LIN {X 0,Y 474.601,Z 136.99,A -85,B 0,C 180,E1 -7407.326,E2 -7407.326} C_VEL
LIN {X 0,Y 474.598,Z 136.978,A -85,B 0,C 180,E1 -7410.231,E2 -7410.231} C_VEL
LIN {X 0,Y 474.615,Z 136.966,A -85,B 0,C 180,E1 -7413.222,E2 -7413.222} C_VEL
LIN {X 0,Y 474.584,Z 136.991,A -85,B 0,C 180,E1 -7416.324,E2 -7416.324} C_VEL
LIN {X 0,Y 474.622,Z 136.969,A -85,B 0,C 180,E1 -7419.548,E2 -7419.548} C_VEL
LIN {X 0,Y 474.577,Z 136.989,A -85,B 0,C 180,E1 -7422.23,E2 -7422.23} C_VEL
LIN {X 0,Y 474.616,Z 136.982,A -85,B 0,C 180,E1 -7425.298,E2 -7425.298} C_VEL
LIN {X 0,Y 474.592,Z 136.991,A -85,B 0,C 180,E1 -7428.211,E2 -7428.211} C_VEL
LIN {X 0,Y 474.608,Z 136.991,A -85,B 0,C 180,E1 -7431.542,E2 -7431.542} C_VEL
LIN {X 0,Y 474.617,Z 136.989,A -85,B 0,C 180,E1 -7434.725,E2 -7434.725} C_VEL
LIN {X 0,Y 474.629,Z 136.988,A -85,B 0,C 180,E1 -7437.787,E2 -7437.787} C_VEL
LIN {X 0,Y 474.575,Z 136.983,A -85,B 0,C 180,E1 -7440.896,E2 -7440.896} C_VEL
LIN {X 0,Y 474.643,Z 137.123,A -85,B 0,C 180,E1 -7442.017,E2 -7442.017} C_VEL
LIN {X 0,Y 477.053,Z 147.679,A -85,B 0,C 180,E1 -7443.983,E2 -7443.983} C_VEL
LIN {X 0,Y 478.463,Z 154.908,A -85,B 0,C 180,E1 -7445.252,E2 -7445.252} C_VEL
LIN {X 0,Y 478.125,Z 161.386,A -85,B 0,C 180,E1 -7446.26,E2 -7446.26} C_VEL
LIN {X 0,Y 479.797,Z 169.232,A -85,B 0,C 180,E1 -7446.509,E2 -7446.509} C_VEL
LIN {X 0,Y 482.553,Z 182.514,A -85,B 0,C 180,E1 -7446.862,E2 -7446.862} C_VEL
LIN {X 0,Y 482.481,Z 187.574,A -85,B 0,C 180,E1 -7446.939,E2 -7446.939} C_VEL
LIN {X 0,Y 481.775,Z 193.424,A -85,B 0,C 180,E1 -7446.996,E2 -7446.996} C_VEL
LIN {X 0,Y 476.297,Z 212.491,A -85,B 0,C 180,E1 -7447.021,E2 -7447.021} C_VEL
LIN {X 0,Y 475.613,Z 218.341,A -85,B 0,C 180,E1 -7447.08,E2 -7447.08} C_VEL
LIN {X 0,Y 474.357,Z 326.967,A -85,B 0,C 180,E1 -7448.779,E2 -7448.779} C_VEL
LIN {X 0,Y 473.824,Z 342.596,A -85,B 0,C 180,E1 -7449.193,E2 -7449.193} C_VEL
LIN {X 0,Y 473.371,Z 356.882,A -85,B 0,C 180,E1 -7449.749,E2 -7449.749} C_VEL
LIN {X 0,Y 472.578,Z 370.807,A -85,B 0,C 180,E1 -7450.451,E2 -7450.451} C_VEL
LIN {X 0,Y 471.793,Z 384.429,A -85,B 0,C 180,E1 -7451.321,E2 -7451.321} C_VEL
LIN {X 0,Y 470.896,Z 396.958,A -85,B 0,C 180,E1 -7452.296,E2 -7452.296} C_VEL
LIN {X 0,Y 470.076,Z 409.646,A -85,B 0,C 180,E1 -7453.497,E2 -7453.497} C_VEL
LIN {X 0,Y 469.269,Z 421.151,A -85,B 0,C 180,E1 -7454.806,E2 -7454.806} C_VEL
LIN {X 0,Y 468.595,Z 430.834,A -85,B 0,C 180,E1 -7456.115,E2 -7456.115} C_VEL
LIN {X 0,Y 467.975,Z 440.24,A -85,B 0,C 180,E1 -7457.627,E2 -7457.627} C_VEL
LIN {X 0,Y 467.546,Z 448.231,A -85,B 0,C 180,E1 -7459.17,E2 -7459.17} C_VEL
LIN {X 0,Y 467.105,Z 455.613,A -85,B 0,C 180,E1 -7460.91,E2 -7460.91} C_VEL
LIN {X 0,Y 466.844,Z 461.472,A -85,B 0,C 180,E1 -7462.648,E2 -7462.648} C_VEL
LIN {X 0,Y 466.79,Z 464.941,A -85,B 0,C 180,E1 -7463.95,E2 -7463.95} C_VEL
LIN {X 0,Y 466.625,Z 468.461,A -85,B 0,C 180,E1 -7465.681,E2 -7465.681} C_VEL
LIN {X 0,Y 466.657,Z 470.79,A -85,B 0,C 180,E1 -7467.41,E2 -7467.41} C_VEL
LIN {X 0,Y 466.587,Z 471.982,A -85,B 0,C 180,E1 -7469.137,E2 -7469.137} C_VEL
LIN {X 0,Y 466.587,Z 472,A -85,B 0,C 180,E1 -7470.863,E2 -7470.863} C_VEL
LIN {X 0,Y 466.658,Z 470.878,A -85,B 0,C 180,E1 -7472.59,E2 -7472.59} C_VEL
LIN {X 0,Y 466.624,Z 468.618,A -85,B 0,C 180,E1 -7474.319,E2 -7474.319} C_VEL
LIN {X 0,Y 466.763,Z 465.163,A -85,B 0,C 180,E1 -7476.05,E2 -7476.05} C_VEL
LIN {X 0,Y 466.909,Z 460.435,A -85,B 0,C 180,E1 -7477.786,E2 -7477.786} C_VEL
LIN {X 0,Y 467.191,Z 454.309,A -85,B 0,C 180,E1 -7479.525,E2 -7479.525} C_VEL
LIN {X 0,Y 467.659,Z 446.597,A -85,B 0,C 180,E1 -7481.266,E2 -7481.266} C_VEL
LIN {X 0,Y 468.093,Z 438.528,A -85,B 0,C 180,E1 -7482.768,E2 -7482.768} C_VEL
LIN {X 0,Y 468.775,Z 428.476,A -85,B 0,C 180,E1 -7484.322,E2 -7484.322} C_VEL
LIN {X 0,Y 469.43,Z 418.327,A -85,B 0,C 180,E1 -7485.634,E2 -7485.634} C_VEL
LIN {X 0,Y 470.225,Z 407.623,A -85,B 0,C 180,E1 -7486.801,E2 -7486.801} C_VEL
LIN {X 0,Y 471.044,Z 395.428,A -85,B 0,C 180,E1 -7487.922,E2 -7487.922} C_VEL
LIN {X 0,Y 471.888,Z 382.566,A -85,B 0,C 180,E1 -7488.901,E2 -7488.901} C_VEL
LIN {X 0,Y 472.684,Z 368.463,A -85,B 0,C 180,E1 -7489.771,E2 -7489.771} C_VEL
LIN {X 0,Y 473.487,Z 353.414,A -85,B 0,C 180,E1 -7490.489,E2 -7490.489} C_VEL
LIN {X 0,Y 473.958,Z 339.526,A -85,B 0,C 180,E1 -7490.99,E2 -7490.99} C_VEL
LIN {X 0,Y 474.358,Z 325.557,A -85,B 0,C 180,E1 -7491.341,E2 -7491.341} C_VEL
LIN {X 0,Y 476.011,Z 183.2,A -85,B 0,C 180,E1 -7493.558,E2 -7493.558} C_VEL
LIN {X 0,Y 471.382,Z 161.527,A -85,B 0,C 180,E1 -7494.186,E2 -7494.186} C_VEL
LIN {X 0,Y 471.552,Z 155.541,A -85,B 0,C 180,E1 -7495.136,E2 -7495.136} C_VEL
LIN {X 0,Y 468.023,Z 139.951,A -85,B 0,C 180,E1 -7497.986,E2 -7497.986} C_VEL
LIN {X 0,Y 467.569,Z 137.908,A -85,B 0,C 180,E1 -7498.444,E2 -7498.444} C_VEL
LIN {X 0,Y 467.546,Z 137.867,A -85,B 0,C 180,E1 -7501.743,E2 -7501.743} C_VEL
LIN {X 0,Y 467.551,Z 137.87,A -85,B 0,C 180,E1 -7504.834,E2 -7504.834} C_VEL
LIN {X 0,Y 467.541,Z 137.87,A -85,B 0,C 180,E1 -7508.047,E2 -7508.047} C_VEL
LIN {X 0,Y 467.561,Z 137.87,A -85,B 0,C 180,E1 -7511.274,E2 -7511.274} C_VEL
LIN {X 0,Y 467.566,Z 137.861,A -85,B 0,C 180,E1 -7514.948,E2 -7514.948} C_VEL
LIN {X 0,Y 467.559,Z 137.858,A -85,B 0,C 180,E1 -7518.595,E2 -7518.595} C_VEL
LIN {X 0,Y 467.552,Z 137.86,A -85,B 0,C 180,E1 -7521.411,E2 -7521.411} C_VEL
LIN {X 0,Y 467.558,Z 137.87,A -85,B 0,C 180,E1 -7524.262,E2 -7524.262} C_VEL
LIN {X 0,Y 467.575,Z 137.84,A -85,B 0,C 180,E1 -7527.323,E2 -7527.323} C_VEL
LIN {X 0,Y 467.552,Z 137.867,A -85,B 0,C 180,E1 -7530.672,E2 -7530.672} C_VEL
LIN {X 0,Y 467.536,Z 137.867,A -85,B 0,C 180,E1 -7533.195,E2 -7533.195} C_VEL
LIN {X 0,Y 467.557,Z 137.865,A -85,B 0,C 180,E1 -7536.056,E2 -7536.056} C_VEL
LIN {X 0,Y 467.621,Z 137.855,A -85,B 0,C 180,E1 -7539.777,E2 -7539.777} C_VEL
LIN {X 0,Y 467.57,Z 137.866,A -85,B 0,C 180,E1 -7542.505,E2 -7542.505} C_VEL
LIN {X 0,Y 467.596,Z 137.855,A -85,B 0,C 180,E1 -7545.196,E2 -7545.196} C_VEL
LIN {X 0,Y 467.659,Z 137.857,A -85,B 0,C 180,E1 -7547.855,E2 -7547.855} C_VEL
LIN {X 0,Y 467.669,Z 137.847,A -85,B 0,C 180,E1 -7551.357,E2 -7551.357} C_VEL
LIN {X 0,Y 467.723,Z 137.849,A -85,B 0,C 180,E1 -7553.962,E2 -7553.962} C_VEL
LIN {X 0,Y 467.824,Z 137.827,A -85,B 0,C 180,E1 -7557.417,E2 -7557.417} C_VEL
LIN {X 0,Y 467.881,Z 137.826,A -85,B 0,C 180,E1 -7560,E2 -7560} C_VEL
LIN {X 0,Y 467.852,Z 137.823,A -85,B 0,C 180,E1 -7562.583,E2 -7562.583} C_VEL
LIN {X 0,Y 467.725,Z 137.845,A -85,B 0,C 180,E1 -7566.038,E2 -7566.038} C_VEL
LIN {X 0,Y 467.671,Z 137.848,A -85,B 0,C 180,E1 -7568.643,E2 -7568.643} C_VEL
LIN {X 0,Y 467.658,Z 137.853,A -85,B 0,C 180,E1 -7572.145,E2 -7572.145} C_VEL
LIN {X 0,Y 467.64,Z 137.85,A -85,B 0,C 180,E1 -7575.695,E2 -7575.695} C_VEL
LIN {X 0,Y 467.623,Z 137.858,A -85,B 0,C 180,E1 -7579.308,E2 -7579.308} C_VEL
LIN {X 0,Y 467.536,Z 137.865,A -85,B 0,C 180,E1 -7582.074,E2 -7582.074} C_VEL
LIN {X 0,Y 467.58,Z 137.863,A -85,B 0,C 180,E1 -7584.889,E2 -7584.889} C_VEL
LIN {X 0,Y 467.618,Z 137.858,A -85,B 0,C 180,E1 -7587.769,E2 -7587.769} C_VEL
LIN {X 0,Y 467.568,Z 137.853,A -85,B 0,C 180,E1 -7591.044,E2 -7591.044} C_VEL
LIN {X 0,Y 467.577,Z 137.846,A -85,B 0,C 180,E1 -7594.24,E2 -7594.24} C_VEL
LIN {X 0,Y 467.549,Z 137.868,A -85,B 0,C 180,E1 -7597.186,E2 -7597.186} C_VEL
LIN {X 0,Y 467.578,Z 137.85,A -85,B 0,C 180,E1 -7600.264,E2 -7600.264} C_VEL
LIN {X 0,Y 467.587,Z 137.866,A -85,B 0,C 180,E1 -7602.567,E2 -7602.567} C_VEL
LIN {X 0,Y 467.567,Z 137.859,A -85,B 0,C 180,E1 -7605.052,E2 -7605.052} C_VEL
LIN {X 0,Y 467.59,Z 137.859,A -85,B 0,C 180,E1 -7607.44,E2 -7607.44} C_VEL
LIN {X 0,Y 467.561,Z 137.861,A -85,B 0,C 180,E1 -7610.853,E2 -7610.853} C_VEL
LIN {X 0,Y 467.56,Z 137.863,A -85,B 0,C 180,E1 -7614.261,E2 -7614.261} C_VEL
LIN {X 0,Y 467.582,Z 137.843,A -85,B 0,C 180,E1 -7617.321,E2 -7617.321} C_VEL
LIN {X 0,Y 467.593,Z 137.978,A -85,B 0,C 180,E1 -7620.582,E2 -7620.582} C_VEL
LIN {X 0,Y 470.698,Z 150.848,A -85,B 0,C 180,E1 -7622.909,E2 -7622.909} C_VEL
LIN {X 0,Y 471.908,Z 156.825,A -85,B 0,C 180,E1 -7623.938,E2 -7623.938} C_VEL
LIN {X 0,Y 471.272,Z 169.442,A -85,B 0,C 180,E1 -7625.859,E2 -7625.859} C_VEL
LIN {X 0,Y 475.948,Z 192.592,A -85,B 0,C 180,E1 -7626.504,E2 -7626.504} C_VEL
LIN {X 0,Y 474.317,Z 332.942,A -85,B 0,C 180,E1 -7628.686,E2 -7628.686} C_VEL
LIN {X 0,Y 473.837,Z 348.179,A -85,B 0,C 180,E1 -7629.062,E2 -7629.062} C_VEL
LIN {X 0,Y 473.282,Z 362.937,A -85,B 0,C 180,E1 -7629.601,E2 -7629.601} C_VEL
LIN {X 0,Y 472.605,Z 375.987,A -85,B 0,C 180,E1 -7630.226,E2 -7630.226} C_VEL
LIN {X 0,Y 471.76,Z 390.279,A -85,B 0,C 180,E1 -7631.094,E2 -7631.094} C_VEL
LIN {X 0,Y 470.911,Z 403.288,A -85,B 0,C 180,E1 -7632.072,E2 -7632.072} C_VEL
LIN {X 0,Y 470.149,Z 414.467,A -85,B 0,C 180,E1 -7633.078,E2 -7633.078} C_VEL
LIN {X 0,Y 469.274,Z 426.416,A -85,B 0,C 180,E1 -7634.361,E2 -7634.361} C_VEL
LIN {X 0,Y 468.65,Z 436.644,A -85,B 0,C 180,E1 -7635.674,E2 -7635.674} C_VEL
LIN {X 0,Y 467.949,Z 446.598,A -85,B 0,C 180,E1 -7637.194,E2 -7637.194} C_VEL
LIN {X 0,Y 467.589,Z 454.94,A -85,B 0,C 180,E1 -7638.732,E2 -7638.732} C_VEL
LIN {X 0,Y 467.104,Z 462.734,A -85,B 0,C 180,E1 -7640.473,E2 -7640.473} C_VEL
LIN {X 0,Y 466.86,Z 468.934,A -85,B 0,C 180,E1 -7642.213,E2 -7642.213} C_VEL
LIN {X 0,Y 466.726,Z 473.728,A -85,B 0,C 180,E1 -7643.949,E2 -7643.949} C_VEL
LIN {X 0,Y 466.601,Z 477.239,A -85,B 0,C 180,E1 -7645.681,E2 -7645.681} C_VEL
LIN {X 0,Y 466.637,Z 479.55,A -85,B 0,C 180,E1 -7647.41,E2 -7647.41} C_VEL
LIN {X 0,Y 466.586,Z 480.712,A -85,B 0,C 180,E1 -7649.137,E2 -7649.137} C_VEL
LIN {X 0,Y 466.586,Z 480.711,A -85,B 0,C 180,E1 -7650.863,E2 -7650.863} C_VEL
LIN {X 0,Y 466.637,Z 479.545,A -85,B 0,C 180,E1 -7652.59,E2 -7652.59} C_VEL
LIN {X 0,Y 466.602,Z 477.233,A -85,B 0,C 180,E1 -7654.319,E2 -7654.319} C_VEL
LIN {X 0,Y 466.751,Z 473.727,A -85,B 0,C 180,E1 -7656.05,E2 -7656.05} C_VEL
LIN {X 0,Y 466.86,Z 468.935,A -85,B 0,C 180,E1 -7657.787,E2 -7657.787} C_VEL
LIN {X 0,Y 467.104,Z 462.726,A -85,B 0,C 180,E1 -7659.527,E2 -7659.527} C_VEL
LIN {X 0,Y 467.588,Z 454.928,A -85,B 0,C 180,E1 -7661.268,E2 -7661.268} C_VEL
LIN {X 0,Y 467.975,Z 446.451,A -85,B 0,C 180,E1 -7662.827,E2 -7662.827} C_VEL
LIN {X 0,Y 468.651,Z 436.633,A -85,B 0,C 180,E1 -7664.326,E2 -7664.326} C_VEL
LIN {X 0,Y 469.301,Z 426.404,A -85,B 0,C 180,E1 -7665.638,E2 -7665.638} C_VEL
LIN {X 0,Y 470.134,Z 414.519,A -85,B 0,C 180,E1 -7666.916,E2 -7666.916} C_VEL
LIN {X 0,Y 470.986,Z 401.979,A -85,B 0,C 180,E1 -7668.037,E2 -7668.037} C_VEL
LIN {X 0,Y 471.834,Z 388.66,A -85,B 0,C 180,E1 -7669.016,E2 -7669.016} C_VEL
LIN {X 0,Y 472.627,Z 375.945,A -85,B 0,C 180,E1 -7669.773,E2 -7669.773} C_VEL
LIN {X 0,Y 473.254,Z 362.971,A -85,B 0,C 180,E1 -7670.397,E2 -7670.397} C_VEL
LIN {X 0,Y 473.858,Z 348.12,A -85,B 0,C 180,E1 -7670.937,E2 -7670.937} C_VEL
LIN {X 0,Y 474.293,Z 332.817,A -85,B 0,C 180,E1 -7671.315,E2 -7671.315} C_VEL
LIN {X 0,Y 475.947,Z 192.412,A -85,B 0,C 180,E1 -7673.496,E2 -7673.496} C_VEL
LIN {X 0,Y 471.259,Z 169.525,A -85,B 0,C 180,E1 -7674.133,E2 -7674.133} C_VEL
LIN {X 0,Y 471.878,Z 156.807,A -85,B 0,C 180,E1 -7676.063,E2 -7676.063} C_VEL
LIN {X 0,Y 469.216,Z 144.362,A -85,B 0,C 180,E1 -7678.23,E2 -7678.23} C_VEL
LIN {X 0,Y 467.581,Z 137.946,A -85,B 0,C 180,E1 -7679.434,E2 -7679.434} C_VEL
LIN {X 0,Y 467.584,Z 137.845,A -85,B 0,C 180,E1 -7682.758,E2 -7682.758} C_VEL
LIN {X 0,Y 467.554,Z 137.864,A -85,B 0,C 180,E1 -7685.89,E2 -7685.89} C_VEL
LIN {X 0,Y 467.561,Z 137.86,A -85,B 0,C 180,E1 -7689.147,E2 -7689.147} C_VEL
LIN {X 0,Y 467.587,Z 137.86,A -85,B 0,C 180,E1 -7692.567,E2 -7692.567} C_VEL
LIN {X 0,Y 467.566,Z 137.86,A -85,B 0,C 180,E1 -7695.053,E2 -7695.053} C_VEL
LIN {X 0,Y 467.589,Z 137.866,A -85,B 0,C 180,E1 -7697.44,E2 -7697.44} C_VEL
LIN {X 0,Y 467.582,Z 137.854,A -85,B 0,C 180,E1 -7700.855,E2 -7700.855} C_VEL
LIN {X 0,Y 467.559,Z 137.862,A -85,B 0,C 180,E1 -7704.261,E2 -7704.261} C_VEL
LIN {X 0,Y 467.574,Z 137.84,A -85,B 0,C 180,E1 -7707.323,E2 -7707.323} C_VEL
LIN {X 0,Y 467.57,Z 137.863,A -85,B 0,C 180,E1 -7710.668,E2 -7710.668} C_VEL
LIN {X 0,Y 467.616,Z 137.858,A -85,B 0,C 180,E1 -7713.2,E2 -7713.2} C_VEL
LIN {X 0,Y 467.594,Z 137.862,A -85,B 0,C 180,E1 -7716.468,E2 -7716.468} C_VEL
LIN {X 0,Y 467.623,Z 137.855,A -85,B 0,C 180,E1 -7719.777,E2 -7719.777} C_VEL
LIN {X 0,Y 467.596,Z 137.863,A -85,B 0,C 180,E1 -7722.506,E2 -7722.506} C_VEL
LIN {X 0,Y 467.606,Z 137.859,A -85,B 0,C 180,E1 -7725.197,E2 -7725.197} C_VEL
LIN {X 0,Y 467.658,Z 137.853,A -85,B 0,C 180,E1 -7727.855,E2 -7727.855} C_VEL
LIN {X 0,Y 467.671,Z 137.849,A -85,B 0,C 180,E1 -7731.357,E2 -7731.357} C_VEL
LIN {X 0,Y 467.725,Z 137.844,A -85,B 0,C 180,E1 -7733.962,E2 -7733.962} C_VEL
LIN {X 0,Y 467.853,Z 137.823,A -85,B 0,C 180,E1 -7737.417,E2 -7737.417} C_VEL
LIN {X 0,Y 467.882,Z 137.826,A -85,B 0,C 180,E1 -7740,E2 -7740} C_VEL
LIN {X 0,Y 467.849,Z 137.824,A -85,B 0,C 180,E1 -7742.583,E2 -7742.583} C_VEL
LIN {X 0,Y 467.723,Z 137.849,A -85,B 0,C 180,E1 -7746.038,E2 -7746.038} C_VEL
LIN {X 0,Y 467.671,Z 137.846,A -85,B 0,C 180,E1 -7748.643,E2 -7748.643} C_VEL
LIN {X 0,Y 467.658,Z 137.858,A -85,B 0,C 180,E1 -7752.145,E2 -7752.145} C_VEL
LIN {X 0,Y 467.63,Z 137.853,A -85,B 0,C 180,E1 -7755.695,E2 -7755.695} C_VEL
LIN {X 0,Y 467.621,Z 137.855,A -85,B 0,C 180,E1 -7759.308,E2 -7759.308} C_VEL
LIN {X 0,Y 467.535,Z 137.874,A -85,B 0,C 180,E1 -7762.074,E2 -7762.074} C_VEL
LIN {X 0,Y 467.561,Z 137.859,A -85,B 0,C 180,E1 -7764.89,E2 -7764.89} C_VEL
LIN {X 0,Y 467.547,Z 137.873,A -85,B 0,C 180,E1 -7767.774,E2 -7767.774} C_VEL
LIN {X 0,Y 467.566,Z 137.851,A -85,B 0,C 180,E1 -7771.044,E2 -7771.044} C_VEL
LIN {X 0,Y 467.577,Z 137.859,A -85,B 0,C 180,E1 -7774.24,E2 -7774.24} C_VEL
LIN {X 0,Y 467.543,Z 137.873,A -85,B 0,C 180,E1 -7777.185,E2 -7777.185} C_VEL
LIN {X 0,Y 467.558,Z 137.845,A -85,B 0,C 180,E1 -7780.267,E2 -7780.267} C_VEL
LIN {X 0,Y 467.545,Z 137.869,A -85,B 0,C 180,E1 -7783.746,E2 -7783.746} C_VEL
LIN {X 0,Y 467.545,Z 137.858,A -85,B 0,C 180,E1 -7786.254,E2 -7786.254} C_VEL
LIN {X 0,Y 467.558,Z 137.859,A -85,B 0,C 180,E1 -7789.733,E2 -7789.733} C_VEL
LIN {X 0,Y 467.542,Z 137.871,A -85,B 0,C 180,E1 -7792.815,E2 -7792.815} C_VEL
LIN {X 0,Y 467.577,Z 137.864,A -85,B 0,C 180,E1 -7795.76,E2 -7795.76} C_VEL
LIN {X 0,Y 467.554,Z 137.869,A -85,B 0,C 180,E1 -7798.258,E2 -7798.258} C_VEL
LIN {X 0,Y 467.577,Z 137.966,A -85,B 0,C 180,E1 -7801.679,E2 -7801.679} C_VEL
LIN {X 0,Y 468.31,Z 140.976,A -85,B 0,C 180,E1 -7802.304,E2 -7802.304} C_VEL
LIN {X 0,Y 471.455,Z 154.975,A -85,B 0,C 180,E1 -7804.859,E2 -7804.859} C_VEL
LIN {X 0,Y 471.458,Z 159.152,A -85,B 0,C 180,E1 -7805.551,E2 -7805.551} C_VEL
LIN {X 0,Y 471.377,Z 161.751,A -85,B 0,C 180,E1 -7805.923,E2 -7805.923} C_VEL
LIN {X 0,Y 476.03,Z 183.831,A -85,B 0,C 180,E1 -7806.546,E2 -7806.546} C_VEL
LIN {X 0,Y 475.613,Z 218.341,A -85,B 0,C 180,E1 -7807.08,E2 -7807.08} C_VEL
LIN {X 0,Y 474.922,Z 224.189,A -85,B 0,C 180,E1 -7807.139,E2 -7807.139} C_VEL
LIN {X 0,Y 469.423,Z 243.244,A -85,B 0,C 180,E1 -7807.165,E2 -7807.165} C_VEL
LIN {X 0,Y 468.75,Z 249.092,A -85,B 0,C 180,E1 -7807.225,E2 -7807.225} C_VEL
LIN {X 0,Y 467.748,Z 327.054,A -85,B 0,C 180,E1 -7808.464,E2 -7808.464} C_VEL
LIN {X 0,Y 467.185,Z 342.973,A -85,B 0,C 180,E1 -7808.894,E2 -7808.894} C_VEL
LIN {X 0,Y 466.691,Z 357.277,A -85,B 0,C 180,E1 -7809.461,E2 -7809.461} C_VEL
LIN {X 0,Y 465.895,Z 370.881,A -85,B 0,C 180,E1 -7810.159,E2 -7810.159} C_VEL
LIN {X 0,Y 465.044,Z 384.502,A -85,B 0,C 180,E1 -7811.039,E2 -7811.039} C_VEL
LIN {X 0,Y 464.123,Z 397.03,A -85,B 0,C 180,E1 -7812.029,E2 -7812.029} C_VEL
LIN {X 0,Y 463.35,Z 408.429,A -85,B 0,C 180,E1 -7813.114,E2 -7813.114} C_VEL
LIN {X 0,Y 462.475,Z 419.444,A -85,B 0,C 180,E1 -7814.351,E2 -7814.351} C_VEL
LIN {X 0,Y 461.775,Z 429.422,A -85,B 0,C 180,E1 -7815.681,E2 -7815.681} C_VEL
LIN {X 0,Y 461.096,Z 438.756,A -85,B 0,C 180,E1 -7817.156,E2 -7817.156} C_VEL
LIN {X 0,Y 460.615,Z 447.293,A -85,B 0,C 180,E1 -7818.782,E2 -7818.782} C_VEL
LIN {X 0,Y 460.157,Z 453.998,A -85,B 0,C 180,E1 -7820.328,E2 -7820.328} C_VEL
LIN {X 0,Y 459.849,Z 460.21,A -85,B 0,C 180,E1 -7822.094,E2 -7822.094} C_VEL
LIN {X 0,Y 459.708,Z 465.009,A -85,B 0,C 180,E1 -7823.857,E2 -7823.857} C_VEL
LIN {X 0,Y 459.544,Z 468.528,A -85,B 0,C 180,E1 -7825.615,E2 -7825.615} C_VEL
LIN {X 0,Y 459.579,Z 470.856,A -85,B 0,C 180,E1 -7827.371,E2 -7827.371} C_VEL
LIN {X 0,Y 459.492,Z 472.049,A -85,B 0,C 180,E1 -7829.124,E2 -7829.124} C_VEL
LIN {X 0,Y 459.492,Z 472.066,A -85,B 0,C 180,E1 -7830.876,E2 -7830.876} C_VEL
LIN {X 0,Y 459.58,Z 470.944,A -85,B 0,C 180,E1 -7832.63,E2 -7832.63} C_VEL
LIN {X 0,Y 459.542,Z 468.683,A -85,B 0,C 180,E1 -7834.386,E2 -7834.386} C_VEL
LIN {X 0,Y 459.665,Z 465.229,A -85,B 0,C 180,E1 -7836.144,E2 -7836.144} C_VEL
LIN {X 0,Y 459.838,Z 460.5,A -85,B 0,C 180,E1 -7837.906,E2 -7837.906} C_VEL
LIN {X 0,Y 460.143,Z 454.374,A -85,B 0,C 180,E1 -7839.672,E2 -7839.672} C_VEL
LIN {X 0,Y 460.646,Z 446.661,A -85,B 0,C 180,E1 -7841.44,E2 -7841.44} C_VEL
LIN {X 0,Y 461.119,Z 438.4,A -85,B 0,C 180,E1 -7842.999,E2 -7842.999} C_VEL
LIN {X 0,Y 461.848,Z 428.539,A -85,B 0,C 180,E1 -7844.542,E2 -7844.542} C_VEL
LIN {X 0,Y 462.537,Z 418.39,A -85,B 0,C 180,E1 -7845.873,E2 -7845.873} C_VEL
LIN {X 0,Y 463.334,Z 408.38,A -85,B 0,C 180,E1 -7846.984,E2 -7846.984} C_VEL
LIN {X 0,Y 464.259,Z 395.49,A -85,B 0,C 180,E1 -7848.193,E2 -7848.193} C_VEL
LIN {X 0,Y 465.161,Z 382.627,A -85,B 0,C 180,E1 -7849.185,E2 -7849.185} C_VEL
LIN {X 0,Y 466.008,Z 368.522,A -85,B 0,C 180,E1 -7850.066,E2 -7850.066} C_VEL
LIN {X 0,Y 466.81,Z 354.384,A -85,B 0,C 180,E1 -7850.755,E2 -7850.755} C_VEL
LIN {X 0,Y 467.28,Z 341.407,A -85,B 0,C 180,E1 -7851.246,E2 -7851.246} C_VEL
LIN {X 0,Y 467.71,Z 327.055,A -85,B 0,C 180,E1 -7851.63,E2 -7851.63} C_VEL
LIN {X 0,Y 469.535,Z 185.525,A -85,B 0,C 180,E1 -7853.866,E2 -7853.866} C_VEL
LIN {X 0,Y 467.636,Z 175.394,A -85,B 0,C 180,E1 -7854.136,E2 -7854.136} C_VEL
LIN {X 0,Y 464.636,Z 161.59,A -85,B 0,C 180,E1 -7854.56,E2 -7854.56} C_VEL
LIN {X 0,Y 464.648,Z 157.026,A -85,B 0,C 180,E1 -7855.296,E2 -7855.296} C_VEL
LIN {X 0,Y 461.438,Z 142.731,A -85,B 0,C 180,E1 -7857.947,E2 -7857.947} C_VEL
LIN {X 0,Y 460.507,Z 138.882,A -85,B 0,C 180,E1 -7858.734,E2 -7858.734} C_VEL
LIN {X 0,Y 460.496,Z 138.734,A -85,B 0,C 180,E1 -7861.277,E2 -7861.277} C_VEL
LIN {X 0,Y 460.52,Z 138.743,A -85,B 0,C 180,E1 -7864.503,E2 -7864.503} C_VEL
LIN {X 0,Y 460.484,Z 138.751,A -85,B 0,C 180,E1 -7867.625,E2 -7867.625} C_VEL
LIN {X 0,Y 460.515,Z 138.744,A -85,B 0,C 180,E1 -7871.013,E2 -7871.013} C_VEL
LIN {X 0,Y 460.512,Z 138.735,A -85,B 0,C 180,E1 -7874.589,E2 -7874.589} C_VEL
LIN {X 0,Y 460.475,Z 138.746,A -85,B 0,C 180,E1 -7877.813,E2 -7877.813} C_VEL
LIN {X 0,Y 460.511,Z 138.723,A -85,B 0,C 180,E1 -7880.135,E2 -7880.135} C_VEL
LIN {X 0,Y 460.472,Z 138.75,A -85,B 0,C 180,E1 -7883.47,E2 -7883.47} C_VEL
LIN {X 0,Y 460.518,Z 138.723,A -85,B 0,C 180,E1 -7886.674,E2 -7886.674} C_VEL
LIN {X 0,Y 460.505,Z 138.731,A -85,B 0,C 180,E1 -7889.759,E2 -7889.759} C_VEL
LIN {X 0,Y 460.493,Z 138.748,A -85,B 0,C 180,E1 -7892.751,E2 -7892.751} C_VEL
LIN {X 0,Y 460.519,Z 138.737,A -85,B 0,C 180,E1 -7895.666,E2 -7895.666} C_VEL
LIN {X 0,Y 460.523,Z 138.74,A -85,B 0,C 180,E1 -7898.578,E2 -7898.578} C_VEL
LIN {X 0,Y 460.584,Z 138.73,A -85,B 0,C 180,E1 -7901.311,E2 -7901.311} C_VEL
LIN {X 0,Y 460.568,Z 138.737,A -85,B 0,C 180,E1 -7904.058,E2 -7904.058} C_VEL
LIN {X 0,Y 460.612,Z 138.732,A -85,B 0,C 180,E1 -7907.666,E2 -7907.666} C_VEL
LIN {X 0,Y 460.619,Z 138.724,A -85,B 0,C 180,E1 -7911.224,E2 -7911.224} C_VEL
LIN {X 0,Y 460.687,Z 138.727,A -85,B 0,C 180,E1 -7913.87,E2 -7913.87} C_VEL
LIN {X 0,Y 460.768,Z 138.706,A -85,B 0,C 180,E1 -7917.377,E2 -7917.377} C_VEL
LIN {X 0,Y 460.85,Z 138.702,A -85,B 0,C 180,E1 -7920,E2 -7920} C_VEL
LIN {X 0,Y 460.793,Z 138.703,A -85,B 0,C 180,E1 -7922.622,E2 -7922.622} C_VEL
LIN {X 0,Y 460.689,Z 138.721,A -85,B 0,C 180,E1 -7926.13,E2 -7926.13} C_VEL
LIN {X 0,Y 460.621,Z 138.727,A -85,B 0,C 180,E1 -7928.776,E2 -7928.776} C_VEL
LIN {X 0,Y 460.616,Z 138.731,A -85,B 0,C 180,E1 -7932.445,E2 -7932.445} C_VEL
LIN {X 0,Y 460.602,Z 138.725,A -85,B 0,C 180,E1 -7935.997,E2 -7935.997} C_VEL
LIN {X 0,Y 460.569,Z 138.733,A -85,B 0,C 180,E1 -7939.615,E2 -7939.615} C_VEL
LIN {X 0,Y 460.512,Z 138.741,A -85,B 0,C 180,E1 -7942.429,E2 -7942.429} C_VEL
LIN {X 0,Y 460.548,Z 138.732,A -85,B 0,C 180,E1 -7945.796,E2 -7945.796} C_VEL
LIN {X 0,Y 460.552,Z 138.74,A -85,B 0,C 180,E1 -7948.233,E2 -7948.233} C_VEL
LIN {X 0,Y 460.521,Z 138.728,A -85,B 0,C 180,E1 -7951.282,E2 -7951.282} C_VEL
LIN {X 0,Y 460.524,Z 138.728,A -85,B 0,C 180,E1 -7954.504,E2 -7954.504} C_VEL
LIN {X 0,Y 460.502,Z 138.745,A -85,B 0,C 180,E1 -7957.623,E2 -7957.623} C_VEL
LIN {X 0,Y 460.543,Z 138.725,A -85,B 0,C 180,E1 -7960.269,E2 -7960.269} C_VEL
LIN {X 0,Y 460.499,Z 138.746,A -85,B 0,C 180,E1 -7963.375,E2 -7963.375} C_VEL
LIN {X 0,Y 460.499,Z 138.738,A -85,B 0,C 180,E1 -7966.624,E2 -7966.624} C_VEL
LIN {X 0,Y 460.54,Z 138.739,A -85,B 0,C 180,E1 -7969.731,E2 -7969.731} C_VEL
LIN {X 0,Y 460.5,Z 138.748,A -85,B 0,C 180,E1 -7972.524,E2 -7972.524} C_VEL
LIN {X 0,Y 460.547,Z 138.745,A -85,B 0,C 180,E1 -7975.624,E2 -7975.624} C_VEL
LIN {X 0,Y 460.538,Z 138.715,A -85,B 0,C 180,E1 -7978.744,E2 -7978.744} C_VEL
LIN {X 0,Y 460.558,Z 138.909,A -85,B 0,C 180,E1 -7980.265,E2 -7980.265} C_VEL
LIN {X 0,Y 463.797,Z 152.276,A -85,B 0,C 180,E1 -7982.717,E2 -7982.717} C_VEL
LIN {X 0,Y 465.079,Z 158.551,A -85,B 0,C 180,E1 -7983.816,E2 -7983.816} C_VEL
LIN {X 0,Y 464.524,Z 169.216,A -85,B 0,C 180,E1 -7985.473,E2 -7985.473} C_VEL
LIN {X 0,Y 469.296,Z 192.542,A -85,B 0,C 180,E1 -7986.15,E2 -7986.15} C_VEL
LIN {X 0,Y 468.69,Z 256.954,A -85,B 0,C 180,E1 -7987.17,E2 -7987.17} C_VEL
LIN {X 0,Y 467.643,Z 335.72,A -85,B 0,C 180,E1 -7988.424,E2 -7988.424} C_VEL
LIN {X 0,Y 467.099,Z 351.363,A -85,B 0,C 180,E1 -7988.852,E2 -7988.852} C_VEL
LIN {X 0,Y 466.503,Z 365.369,A -85,B 0,C 180,E1 -7989.401,E2 -7989.401} C_VEL
LIN {X 0,Y 465.718,Z 379.903,A -85,B 0,C 180,E1 -7990.151,E2 -7990.151} C_VEL
LIN {X 0,Y 464.835,Z 393.382,A -85,B 0,C 180,E1 -7991.03,E2 -7991.03} C_VEL
LIN {X 0,Y 463.954,Z 405.808,A -85,B 0,C 180,E1 -7992.023,E2 -7992.023} C_VEL
LIN {X 0,Y 463.021,Z 418.444,A -85,B 0,C 180,E1 -7993.238,E2 -7993.238} C_VEL
LIN {X 0,Y 462.156,Z 429.922,A -85,B 0,C 180,E1 -7994.566,E2 -7994.566} C_VEL
LIN {X 0,Y 461.482,Z 439.581,A -85,B 0,C 180,E1 -7995.897,E2 -7995.897} C_VEL
LIN {X 0,Y 460.781,Z 449.144,A -85,B 0,C 180,E1 -7997.461,E2 -7997.461} C_VEL
LIN {X 0,Y 460.423,Z 456.966,A -85,B 0,C 180,E1 -7999,E2 -7999} C_VEL
LIN {X 0,Y 459.983,Z 464.339,A -85,B 0,C 180,E1 -8000.768,E2 -8000.768} C_VEL
LIN {X 0,Y 459.747,Z 470.187,A -85,B 0,C 180,E1 -8002.534,E2 -8002.534} C_VEL
LIN {X 0,Y 459.637,Z 473.662,A -85,B 0,C 180,E1 -8003.856,E2 -8003.856} C_VEL
LIN {X 0,Y 459.52,Z 477.173,A -85,B 0,C 180,E1 -8005.614,E2 -8005.614} C_VEL
LIN {X 0,Y 459.559,Z 479.484,A -85,B 0,C 180,E1 -8007.37,E2 -8007.37} C_VEL
LIN {X 0,Y 459.491,Z 480.645,A -85,B 0,C 180,E1 -8009.124,E2 -8009.124} C_VEL
LIN {X 0,Y 459.491,Z 480.644,A -85,B 0,C 180,E1 -8010.876,E2 -8010.876} C_VEL
LIN {X 0,Y 459.559,Z 479.478,A -85,B 0,C 180,E1 -8012.63,E2 -8012.63} C_VEL
LIN {X 0,Y 459.52,Z 477.167,A -85,B 0,C 180,E1 -8014.386,E2 -8014.386} C_VEL
LIN {X 0,Y 459.66,Z 473.66,A -85,B 0,C 180,E1 -8016.144,E2 -8016.144} C_VEL
LIN {X 0,Y 459.799,Z 468.868,A -85,B 0,C 180,E1 -8017.907,E2 -8017.907} C_VEL
LIN {X 0,Y 460.032,Z 462.658,A -85,B 0,C 180,E1 -8019.674,E2 -8019.674} C_VEL
LIN {X 0,Y 460.568,Z 454.86,A -85,B 0,C 180,E1 -8021.442,E2 -8021.442} C_VEL
LIN {X 0,Y 460.988,Z 446.546,A -85,B 0,C 180,E1 -8022.998,E2 -8022.998} C_VEL
LIN {X 0,Y 461.691,Z 436.564,A -85,B 0,C 180,E1 -8024.547,E2 -8024.547} C_VEL
LIN {X 0,Y 462.404,Z 426.335,A -85,B 0,C 180,E1 -8025.877,E2 -8025.877} C_VEL
LIN {X 0,Y 463.362,Z 413.867,A -85,B 0,C 180,E1 -8027.232,E2 -8027.232} C_VEL
LIN {X 0,Y 464.317,Z 400.575,A -85,B 0,C 180,E1 -8028.419,E2 -8028.419} C_VEL
LIN {X 0,Y 465.211,Z 386.964,A -85,B 0,C 180,E1 -8029.412,E2 -8029.412} C_VEL
LIN {X 0,Y 466.127,Z 372.864,A -85,B 0,C 180,E1 -8030.233,E2 -8030.233} C_VEL
LIN {X 0,Y 466.831,Z 357.475,A -85,B 0,C 180,E1 -8030.927,E2 -8030.927} C_VEL
LIN {X 0,Y 467.432,Z 342.455,A -85,B 0,C 180,E1 -8031.412,E2 -8031.412} C_VEL
LIN {X 0,Y 467.813,Z 326.542,A -85,B 0,C 180,E1 -8031.741,E2 -8031.741} C_VEL
LIN {X 0,Y 469.421,Z 193.489,A -85,B 0,C 180,E1 -8033.824,E2 -8033.824} C_VEL
LIN {X 0,Y 464.488,Z 169.332,A -85,B 0,C 180,E1 -8034.516,E2 -8034.516} C_VEL
LIN {X 0,Y 465.073,Z 158.535,A -85,B 0,C 180,E1 -8036.184,E2 -8036.184} C_VEL
LIN {X 0,Y 462.412,Z 146.272,A -85,B 0,C 180,E1 -8038.356,E2 -8038.356} C_VEL
LIN {X 0,Y 460.557,Z 138.835,A -85,B 0,C 180,E1 -8039.759,E2 -8039.759} C_VEL
LIN {X 0,Y 460.531,Z 138.725,A -85,B 0,C 180,E1 -8042.93,E2 -8042.93} C_VEL
LIN {X 0,Y 460.498,Z 138.742,A -85,B 0,C 180,E1 -8046.014,E2 -8046.014} C_VEL
LIN {X 0,Y 460.535,Z 138.736,A -85,B 0,C 180,E1 -8048.896,E2 -8048.896} C_VEL
LIN {X 0,Y 460.523,Z 138.742,A -85,B 0,C 180,E1 -8052.181,E2 -8052.181} C_VEL
LIN {X 0,Y 460.514,Z 138.741,A -85,B 0,C 180,E1 -8055.411,E2 -8055.411} C_VEL
LIN {X 0,Y 460.532,Z 138.732,A -85,B 0,C 180,E1 -8058.398,E2 -8058.398} C_VEL
LIN {X 0,Y 460.526,Z 138.736,A -85,B 0,C 180,E1 -8061.267,E2 -8061.267} C_VEL
LIN {X 0,Y 460.509,Z 138.74,A -85,B 0,C 180,E1 -8064.554,E2 -8064.554} C_VEL
LIN {X 0,Y 460.526,Z 138.72,A -85,B 0,C 180,E1 -8067.715,E2 -8067.715} C_VEL
LIN {X 0,Y 460.54,Z 138.74,A -85,B 0,C 180,E1 -8070.769,E2 -8070.769} C_VEL
LIN {X 0,Y 460.56,Z 138.732,A -85,B 0,C 180,E1 -8073.735,E2 -8073.735} C_VEL
LIN {X 0,Y 460.547,Z 138.741,A -85,B 0,C 180,E1 -8076.624,E2 -8076.624} C_VEL
LIN {X 0,Y 460.552,Z 138.737,A -85,B 0,C 180,E1 -8079.453,E2 -8079.453} C_VEL
LIN {X 0,Y 460.548,Z 138.739,A -85,B 0,C 180,E1 -8082.23,E2 -8082.23} C_VEL
LIN {X 0,Y 460.565,Z 138.733,A -85,B 0,C 180,E1 -8084.965,E2 -8084.965} C_VEL
LIN {X 0,Y 460.612,Z 138.735,A -85,B 0,C 180,E1 -8088.559,E2 -8088.559} C_VEL
LIN {X 0,Y 460.621,Z 138.728,A -85,B 0,C 180,E1 -8091.224,E2 -8091.224} C_VEL
LIN {X 0,Y 460.689,Z 138.721,A -85,B 0,C 180,E1 -8093.87,E2 -8093.87} C_VEL
LIN {X 0,Y 460.793,Z 138.703,A -85,B 0,C 180,E1 -8097.378,E2 -8097.378} C_VEL
LIN {X 0,Y 460.852,Z 138.702,A -85,B 0,C 180,E1 -8100,E2 -8100} C_VEL
LIN {X 0,Y 460.789,Z 138.703,A -85,B 0,C 180,E1 -8102.623,E2 -8102.623} C_VEL
LIN {X 0,Y 460.687,Z 138.726,A -85,B 0,C 180,E1 -8106.13,E2 -8106.13} C_VEL
LIN {X 0,Y 460.621,Z 138.724,A -85,B 0,C 180,E1 -8108.776,E2 -8108.776} C_VEL
LIN {X 0,Y 460.611,Z 138.733,A -85,B 0,C 180,E1 -8112.334,E2 -8112.334} C_VEL
LIN {X 0,Y 460.58,Z 138.735,A -85,B 0,C 180,E1 -8115.988,E2 -8115.988} C_VEL
LIN {X 0,Y 460.568,Z 138.734,A -85,B 0,C 180,E1 -8119.616,E2 -8119.616} C_VEL
LIN {X 0,Y 460.512,Z 138.745,A -85,B 0,C 180,E1 -8122.429,E2 -8122.429} C_VEL
LIN {X 0,Y 460.536,Z 138.738,A -85,B 0,C 180,E1 -8125.793,E2 -8125.793} C_VEL
LIN {X 0,Y 460.521,Z 138.744,A -85,B 0,C 180,E1 -8129.232,E2 -8129.232} C_VEL
LIN {X 0,Y 460.519,Z 138.715,A -85,B 0,C 180,E1 -8132.285,E2 -8132.285} C_VEL
LIN {X 0,Y 460.507,Z 138.746,A -85,B 0,C 180,E1 -8135.446,E2 -8135.446} C_VEL
LIN {X 0,Y 460.504,Z 138.736,A -85,B 0,C 180,E1 -8138.891,E2 -8138.891} C_VEL
LIN {X 0,Y 460.502,Z 138.737,A -85,B 0,C 180,E1 -8141.598,E2 -8141.598} C_VEL
LIN {X 0,Y 460.512,Z 138.744,A -85,B 0,C 180,E1 -8144.589,E2 -8144.589} C_VEL
LIN {X 0,Y 460.476,Z 138.75,A -85,B 0,C 180,E1 -8147.813,E2 -8147.813} C_VEL
LIN {X 0,Y 460.513,Z 138.736,A -85,B 0,C 180,E1 -8150.136,E2 -8150.136} C_VEL
LIN {X 0,Y 460.472,Z 138.745,A -85,B 0,C 180,E1 -8153.47,E2 -8153.47} C_VEL
LIN {X 0,Y 460.519,Z 138.742,A -85,B 0,C 180,E1 -8156.674,E2 -8156.674} C_VEL
LIN {X 0,Y 460.479,Z 138.727,A -85,B 0,C 180,E1 -8159.758,E2 -8159.758} C_VEL
LIN {X 0,Y 460.527,Z 138.948,A -85,B 0,C 180,E1 -8161.392,E2 -8161.392} C_VEL
LIN {X 0,Y 463.164,Z 150.156,A -85,B 0,C 180,E1 -8163.542,E2 -8163.542} C_VEL
LIN {X 0,Y 464.796,Z 157.883,A -85,B 0,C 180,E1 -8164.952,E2 -8164.952} C_VEL
LIN {X 0,Y 464.634,Z 161.858,A -85,B 0,C 180,E1 -8165.553,E2 -8165.553} C_VEL
LIN {X 0,Y 469.521,Z 184.299,A -85,B 0,C 180,E1 -8166.207,E2 -8166.207} C_VEL
LIN {X 0,Y 468.75,Z 249.092,A -85,B 0,C 180,E1 -8167.225,E2 -8167.225} C_VEL
LIN {X 0,Y 468.087,Z 254.938,A -85,B 0,C 180,E1 -8167.286,E2 -8167.286} C_VEL
LIN {X 0,Y 462.579,Z 273.995,A -85,B 0,C 180,E1 -8167.314,E2 -8167.314} C_VEL
LIN {X 0,Y 461.823,Z 279.846,A -85,B 0,C 180,E1 -8167.371,E2 -8167.371} C_VEL
LIN {X 0,Y 461.122,Z 328.065,A -85,B 0,C 180,E1 -8168.162,E2 -8168.162} C_VEL
LIN {X 0,Y 460.566,Z 343.14,A -85,B 0,C 180,E1 -8168.58,E2 -8168.58} C_VEL
LIN {X 0,Y 460.032,Z 357.701,A -85,B 0,C 180,E1 -8169.166,E2 -8169.166} C_VEL
LIN {X 0,Y 459.209,Z 370.955,A -85,B 0,C 180,E1 -8169.858,E2 -8169.858} C_VEL
LIN {X 0,Y 458.315,Z 384.575,A -85,B 0,C 180,E1 -8170.75,E2 -8170.75} C_VEL
LIN {X 0,Y 457.342,Z 397.102,A -85,B 0,C 180,E1 -8171.754,E2 -8171.754} C_VEL
LIN {X 0,Y 456.401,Z 409.788,A -85,B 0,C 180,E1 -8172.988,E2 -8172.988} C_VEL
LIN {X 0,Y 455.484,Z 421.291,A -85,B 0,C 180,E1 -8174.335,E2 -8174.335} C_VEL
LIN {X 0,Y 454.734,Z 430.974,A -85,B 0,C 180,E1 -8175.683,E2 -8175.683} C_VEL
LIN {X 0,Y 453.998,Z 440.313,A -85,B 0,C 180,E1 -8177.228,E2 -8177.228} C_VEL
LIN {X 0,Y 453.542,Z 448.368,A -85,B 0,C 180,E1 -8178.831,E2 -8178.831} C_VEL
LIN {X 0,Y 453.023,Z 455.749,A -85,B 0,C 180,E1 -8180.625,E2 -8180.625} C_VEL
LIN {X 0,Y 452.713,Z 461.608,A -85,B 0,C 180,E1 -8182.417,E2 -8182.417} C_VEL
LIN {X 0,Y 452.632,Z 465.077,A -85,B 0,C 180,E1 -8183.76,E2 -8183.76} C_VEL
LIN {X 0,Y 452.465,Z 468.595,A -85,B 0,C 180,E1 -8185.546,E2 -8185.546} C_VEL
LIN {X 0,Y 452.503,Z 470.923,A -85,B 0,C 180,E1 -8187.329,E2 -8187.329} C_VEL
LIN {X 0,Y 452.401,Z 472.115,A -85,B 0,C 180,E1 -8189.11,E2 -8189.11} C_VEL
LIN {X 0,Y 452.401,Z 472.132,A -85,B 0,C 180,E1 -8190.89,E2 -8190.89} C_VEL
LIN {X 0,Y 452.503,Z 471.009,A -85,B 0,C 180,E1 -8192.671,E2 -8192.671} C_VEL
LIN {X 0,Y 452.463,Z 468.749,A -85,B 0,C 180,E1 -8194.454,E2 -8194.454} C_VEL
LIN {X 0,Y 452.582,Z 465.001,A -85,B 0,C 180,E1 -8196.364,E2 -8196.364} C_VEL
LIN {X 0,Y 452.788,Z 460.565,A -85,B 0,C 180,E1 -8198.03,E2 -8198.03} C_VEL
LIN {X 0,Y 453.103,Z 454.439,A -85,B 0,C 180,E1 -8199.824,E2 -8199.824} C_VEL
LIN {X 0,Y 453.642,Z 446.726,A -85,B 0,C 180,E1 -8201.619,E2 -8201.619} C_VEL
LIN {X 0,Y 454.136,Z 438.492,A -85,B 0,C 180,E1 -8203.197,E2 -8203.197} C_VEL
LIN {X 0,Y 454.912,Z 428.603,A -85,B 0,C 180,E1 -8204.768,E2 -8204.768} C_VEL
LIN {X 0,Y 455.658,Z 418.454,A -85,B 0,C 180,E1 -8206.119,E2 -8206.119} C_VEL
LIN {X 0,Y 456.579,Z 407.188,A -85,B 0,C 180,E1 -8207.379,E2 -8207.379} C_VEL
LIN {X 0,Y 457.594,Z 394.263,A -85,B 0,C 180,E1 -8208.584,E2 -8208.584} C_VEL
LIN {X 0,Y 458.525,Z 381.108,A -85,B 0,C 180,E1 -8209.59,E2 -8209.59} C_VEL
LIN {X 0,Y 459.344,Z 368.58,A -85,B 0,C 180,E1 -8210.37,E2 -8210.37} C_VEL
LIN {X 0,Y 460.164,Z 353.854,A -85,B 0,C 180,E1 -8211.095,E2 -8211.095} C_VEL
LIN {X 0,Y 460.707,Z 340.544,A -85,B 0,C 180,E1 -8211.594,E2 -8211.594} C_VEL
LIN {X 0,Y 461.161,Z 325.643,A -85,B 0,C 180,E1 -8211.983,E2 -8211.983} C_VEL
LIN {X 0,Y 463.05,Z 185.856,A -85,B 0,C 180,E1 -8214.216,E2 -8214.216} C_VEL
LIN {X 0,Y 457.911,Z 161.907,A -85,B 0,C 180,E1 -8214.929,E2 -8214.929} C_VEL
LIN {X 0,Y 457.929,Z 160.498,A -85,B 0,C 180,E1 -8215.11,E2 -8215.11} C_VEL
LIN {X 0,Y 456.853,Z 154.257,A -85,B 0,C 180,E1 -8216.249,E2 -8216.249} C_VEL
LIN {X 0,Y 453.887,Z 141.495,A -85,B 0,C 180,E1 -8218.686,E2 -8218.686} C_VEL
LIN {X 0,Y 453.463,Z 139.681,A -85,B 0,C 180,E1 -8219.111,E2 -8219.111} C_VEL
LIN {X 0,Y 453.442,Z 139.623,A -85,B 0,C 180,E1 -8221.801,E2 -8221.801} C_VEL
LIN {X 0,Y 453.473,Z 139.626,A -85,B 0,C 180,E1 -8224.99,E2 -8224.99} C_VEL
LIN {X 0,Y 453.445,Z 139.627,A -85,B 0,C 180,E1 -8228.314,E2 -8228.314} C_VEL
LIN {X 0,Y 453.47,Z 139.615,A -85,B 0,C 180,E1 -8230.612,E2 -8230.612} C_VEL
LIN {X 0,Y 453.482,Z 139.61,A -85,B 0,C 180,E1 -8234.528,E2 -8234.528} C_VEL
LIN {X 0,Y 453.437,Z 139.624,A -85,B 0,C 180,E1 -8238.071,E2 -8238.071} C_VEL
LIN {X 0,Y 453.444,Z 139.607,A -85,B 0,C 180,E1 -8240.801,E2 -8240.801} C_VEL
LIN {X 0,Y 453.451,Z 139.625,A -85,B 0,C 180,E1 -8243.917,E2 -8243.917} C_VEL
LIN {X 0,Y 453.475,Z 139.595,A -85,B 0,C 180,E1 -8247.15,E2 -8247.15} C_VEL
LIN {X 0,Y 453.463,Z 139.613,A -85,B 0,C 180,E1 -8250.267,E2 -8250.267} C_VEL
LIN {X 0,Y 453.443,Z 139.623,A -85,B 0,C 180,E1 -8253.29,E2 -8253.29} C_VEL
LIN {X 0,Y 453.494,Z 139.618,A -85,B 0,C 180,E1 -8256.238,E2 -8256.238} C_VEL
LIN {X 0,Y 453.482,Z 139.614,A -85,B 0,C 180,E1 -8259.118,E2 -8259.118} C_VEL
LIN {X 0,Y 453.489,Z 139.62,A -85,B 0,C 180,E1 -8261.944,E2 -8261.944} C_VEL
LIN {X 0,Y 453.522,Z 139.607,A -85,B 0,C 180,E1 -8264.726,E2 -8264.726} C_VEL
LIN {X 0,Y 453.561,Z 139.611,A -85,B 0,C 180,E1 -8268.379,E2 -8268.379} C_VEL
LIN {X 0,Y 453.586,Z 139.6,A -85,B 0,C 180,E1 -8271.086,E2 -8271.086} C_VEL
LIN {X 0,Y 453.653,Z 139.602,A -85,B 0,C 180,E1 -8273.774,E2 -8273.774} C_VEL
LIN {X 0,Y 453.715,Z 139.584,A -85,B 0,C 180,E1 -8277.336,E2 -8277.336} C_VEL
LIN {X 0,Y 453.82,Z 139.578,A -85,B 0,C 180,E1 -8280,E2 -8280} C_VEL
LIN {X 0,Y 453.737,Z 139.581,A -85,B 0,C 180,E1 -8282.663,E2 -8282.663} C_VEL
LIN {X 0,Y 453.655,Z 139.597,A -85,B 0,C 180,E1 -8286.226,E2 -8286.226} C_VEL
LIN {X 0,Y 453.587,Z 139.604,A -85,B 0,C 180,E1 -8288.913,E2 -8288.913} C_VEL
LIN {X 0,Y 453.566,Z 139.61,A -85,B 0,C 180,E1 -8292.529,E2 -8292.529} C_VEL
LIN {X 0,Y 453.546,Z 139.604,A -85,B 0,C 180,E1 -8296.196,E2 -8296.196} C_VEL
LIN {X 0,Y 453.518,Z 139.618,A -85,B 0,C 180,E1 -8299.039,E2 -8299.039} C_VEL
LIN {X 0,Y 453.478,Z 139.615,A -85,B 0,C 180,E1 -8301.836,E2 -8301.836} C_VEL
LIN {X 0,Y 453.497,Z 139.62,A -85,B 0,C 180,E1 -8304.735,E2 -8304.735} C_VEL
LIN {X 0,Y 453.531,Z 139.613,A -85,B 0,C 180,E1 -8307.959,E2 -8307.959} C_VEL
LIN {X 0,Y 453.465,Z 139.605,A -85,B 0,C 180,E1 -8311.524,E2 -8311.524} C_VEL
LIN {X 0,Y 453.483,Z 139.609,A -85,B 0,C 180,E1 -8314.776,E2 -8314.776} C_VEL
LIN {X 0,Y 453.465,Z 139.621,A -85,B 0,C 180,E1 -8318.311,E2 -8318.311} C_VEL
LIN {X 0,Y 453.495,Z 139.602,A -85,B 0,C 180,E1 -8320.609,E2 -8320.609} C_VEL
LIN {X 0,Y 453.455,Z 139.624,A -85,B 0,C 180,E1 -8323.244,E2 -8323.244} C_VEL
LIN {X 0,Y 453.464,Z 139.612,A -85,B 0,C 180,E1 -8325.779,E2 -8325.779} C_VEL
LIN {X 0,Y 453.48,Z 139.625,A -85,B 0,C 180,E1 -8328.209,E2 -8328.209} C_VEL
LIN {X 0,Y 453.488,Z 139.612,A -85,B 0,C 180,E1 -8330.794,E2 -8330.794} C_VEL
LIN {X 0,Y 453.455,Z 139.619,A -85,B 0,C 180,E1 -8333.917,E2 -8333.917} C_VEL
LIN {X 0,Y 453.483,Z 139.599,A -85,B 0,C 180,E1 -8337.151,E2 -8337.151} C_VEL
LIN {X 0,Y 453.522,Z 139.788,A -85,B 0,C 180,E1 -8339.918,E2 -8339.918} C_VEL
LIN {X 0,Y 456.593,Z 152.3,A -85,B 0,C 180,E1 -8342.265,E2 -8342.265} C_VEL
LIN {X 0,Y 458.166,Z 159.682,A -85,B 0,C 180,E1 -8343.587,E2 -8343.587} C_VEL
LIN {X 0,Y 457.757,Z 169.158,A -85,B 0,C 180,E1 -8345.086,E2 -8345.086} C_VEL
LIN {X 0,Y 462.043,Z 189.914,A -85,B 0,C 180,E1 -8345.709,E2 -8345.709} C_VEL
LIN {X 0,Y 462.927,Z 194.577,A -85,B 0,C 180,E1 -8345.836,E2 -8345.836} C_VEL
LIN {X 0,Y 461.104,Z 334.344,A -85,B 0,C 180,E1 -8348.073,E2 -8348.073} C_VEL
LIN {X 0,Y 460.55,Z 349.895,A -85,B 0,C 180,E1 -8348.487,E2 -8348.487} C_VEL
LIN {X 0,Y 459.912,Z 364.317,A -85,B 0,C 180,E1 -8349.048,E2 -8349.048} C_VEL
LIN {X 0,Y 459.111,Z 377.853,A -85,B 0,C 180,E1 -8349.736,E2 -8349.736} C_VEL
LIN {X 0,Y 458.15,Z 391.736,A -85,B 0,C 180,E1 -8350.626,E2 -8350.626} C_VEL
LIN {X 0,Y 457.238,Z 404.452,A -85,B 0,C 180,E1 -8351.633,E2 -8351.633} C_VEL
LIN {X 0,Y 456.348,Z 415.856,A -85,B 0,C 180,E1 -8352.714,E2 -8352.714} C_VEL
LIN {X 0,Y 455.534,Z 426.286,A -85,B 0,C 180,E1 -8353.877,E2 -8353.877} C_VEL
LIN {X 0,Y 454.75,Z 436.513,A -85,B 0,C 180,E1 -8355.226,E2 -8355.226} C_VEL
LIN {X 0,Y 453.983,Z 446.641,A -85,B 0,C 180,E1 -8356.823,E2 -8356.823} C_VEL
LIN {X 0,Y 453.549,Z 454.809,A -85,B 0,C 180,E1 -8358.379,E2 -8358.379} C_VEL
LIN {X 0,Y 452.969,Z 462.602,A -85,B 0,C 180,E1 -8360.173,E2 -8360.173} C_VEL
LIN {X 0,Y 452.727,Z 468.802,A -85,B 0,C 180,E1 -8361.969,E2 -8361.969} C_VEL
LIN {X 0,Y 452.562,Z 473.596,A -85,B 0,C 180,E1 -8363.759,E2 -8363.759} C_VEL
LIN {X 0,Y 452.44,Z 477.107,A -85,B 0,C 180,E1 -8365.545,E2 -8365.545} C_VEL
LIN {X 0,Y 452.482,Z 479.418,A -85,B 0,C 180,E1 -8367.329,E2 -8367.329} C_VEL
LIN {X 0,Y 452.4,Z 480.579,A -85,B 0,C 180,E1 -8369.11,E2 -8369.11} C_VEL
LIN {X 0,Y 452.4,Z 480.578,A -85,B 0,C 180,E1 -8370.89,E2 -8370.89} C_VEL
LIN {X 0,Y 452.482,Z 479.412,A -85,B 0,C 180,E1 -8372.671,E2 -8372.671} C_VEL
LIN {X 0,Y 452.441,Z 477.1,A -85,B 0,C 180,E1 -8374.454,E2 -8374.454} C_VEL
LIN {X 0,Y 452.608,Z 473.222,A -85,B 0,C 180,E1 -8376.396,E2 -8376.396} C_VEL
LIN {X 0,Y 452.727,Z 468.8,A -85,B 0,C 180,E1 -8378.031,E2 -8378.031} C_VEL
LIN {X 0,Y 452.969,Z 462.59,A -85,B 0,C 180,E1 -8379.827,E2 -8379.827} C_VEL
LIN {X 0,Y 453.531,Z 454.791,A -85,B 0,C 180,E1 -8381.622,E2 -8381.622} C_VEL
LIN {X 0,Y 453.989,Z 446.626,A -85,B 0,C 180,E1 -8383.176,E2 -8383.176} C_VEL
LIN {X 0,Y 454.754,Z 436.495,A -85,B 0,C 180,E1 -8384.774,E2 -8384.774} C_VEL
LIN {X 0,Y 455.534,Z 426.266,A -85,B 0,C 180,E1 -8386.123,E2 -8386.123} C_VEL
LIN {X 0,Y 456.491,Z 414.258,A -85,B 0,C 180,E1 -8387.451,E2 -8387.451} C_VEL
LIN {X 0,Y 457.441,Z 401.839,A -85,B 0,C 180,E1 -8388.59,E2 -8388.59} C_VEL
LIN {X 0,Y 458.386,Z 388.519,A -85,B 0,C 180,E1 -8389.596,E2 -8389.596} C_VEL
LIN {X 0,Y 459.402,Z 373.815,A -85,B 0,C 180,E1 -8390.484,E2 -8390.484} C_VEL
LIN {X 0,Y 460.139,Z 359.054,A -85,B 0,C 180,E1 -8391.176,E2 -8391.176} C_VEL
LIN {X 0,Y 460.751,Z 344.303,A -85,B 0,C 180,E1 -8391.68,E2 -8391.68} C_VEL
LIN {X 0,Y 461.176,Z 329.643,A -85,B 0,C 180,E1 -8392.011,E2 -8392.011} C_VEL
LIN {X 0,Y 462.945,Z 194.648,A -85,B 0,C 180,E1 -8394.158,E2 -8394.158} C_VEL
LIN {X 0,Y 457.73,Z 169.198,A -85,B 0,C 180,E1 -8394.907,E2 -8394.907} C_VEL
LIN {X 0,Y 458.161,Z 159.654,A -85,B 0,C 180,E1 -8396.414,E2 -8396.414} C_VEL
LIN {X 0,Y 455.129,Z 146.197,A -85,B 0,C 180,E1 -8398.852,E2 -8398.852} C_VEL
LIN {X 0,Y 453.491,Z 139.724,A -85,B 0,C 180,E1 -8400.102,E2 -8400.102} C_VEL
LIN {X 0,Y 453.491,Z 139.606,A -85,B 0,C 180,E1 -8403.189,E2 -8403.189} C_VEL
LIN {X 0,Y 453.453,Z 139.62,A -85,B 0,C 180,E1 -8406.299,E2 -8406.299} C_VEL
LIN {X 0,Y 453.484,Z 139.612,A -85,B 0,C 180,E1 -8409.45,E2 -8409.45} C_VEL
LIN {X 0,Y 453.477,Z 139.623,A -85,B 0,C 180,E1 -8411.935,E2 -8411.935} C_VEL
LIN {X 0,Y 453.485,Z 139.617,A -85,B 0,C 180,E1 -8415.471,E2 -8415.471} C_VEL
LIN {X 0,Y 453.479,Z 139.611,A -85,B 0,C 180,E1 -8418.209,E2 -8418.209} C_VEL
LIN {X 0,Y 453.495,Z 139.608,A -85,B 0,C 180,E1 -8420.793,E2 -8420.793} C_VEL
LIN {X 0,Y 453.454,Z 139.621,A -85,B 0,C 180,E1 -8423.917,E2 -8423.917} C_VEL
LIN {X 0,Y 453.474,Z 139.593,A -85,B 0,C 180,E1 -8427.151,E2 -8427.151} C_VEL
LIN {X 0,Y 453.475,Z 139.618,A -85,B 0,C 180,E1 -8430.268,E2 -8430.268} C_VEL
LIN {X 0,Y 453.505,Z 139.613,A -85,B 0,C 180,E1 -8433.294,E2 -8433.294} C_VEL
LIN {X 0,Y 453.503,Z 139.617,A -85,B 0,C 180,E1 -8436.239,E2 -8436.239} C_VEL
LIN {X 0,Y 453.483,Z 139.615,A -85,B 0,C 180,E1 -8439.118,E2 -8439.118} C_VEL
LIN {X 0,Y 453.502,Z 139.616,A -85,B 0,C 180,E1 -8441.944,E2 -8441.944} C_VEL
LIN {X 0,Y 453.54,Z 139.606,A -85,B 0,C 180,E1 -8444.726,E2 -8444.726} C_VEL
LIN {X 0,Y 453.561,Z 139.612,A -85,B 0,C 180,E1 -8448.379,E2 -8448.379} C_VEL
LIN {X 0,Y 453.587,Z 139.603,A -85,B 0,C 180,E1 -8451.087,E2 -8451.087} C_VEL
LIN {X 0,Y 453.654,Z 139.597,A -85,B 0,C 180,E1 -8453.774,E2 -8453.774} C_VEL
LIN {X 0,Y 453.737,Z 139.582,A -85,B 0,C 180,E1 -8457.337,E2 -8457.337} C_VEL
LIN {X 0,Y 453.821,Z 139.577,A -85,B 0,C 180,E1 -8460,E2 -8460} C_VEL
LIN {X 0,Y 453.732,Z 139.581,A -85,B 0,C 180,E1 -8462.663,E2 -8462.663} C_VEL
LIN {X 0,Y 453.653,Z 139.603,A -85,B 0,C 180,E1 -8466.226,E2 -8466.226} C_VEL
LIN {X 0,Y 453.587,Z 139.6,A -85,B 0,C 180,E1 -8468.914,E2 -8468.914} C_VEL
LIN {X 0,Y 453.566,Z 139.608,A -85,B 0,C 180,E1 -8472.529,E2 -8472.529} C_VEL
LIN {X 0,Y 453.538,Z 139.615,A -85,B 0,C 180,E1 -8476.196,E2 -8476.196} C_VEL
LIN {X 0,Y 453.518,Z 139.61,A -85,B 0,C 180,E1 -8479.039,E2 -8479.039} C_VEL
LIN {X 0,Y 453.478,Z 139.622,A -85,B 0,C 180,E1 -8481.836,E2 -8481.836} C_VEL
LIN {X 0,Y 453.471,Z 139.614,A -85,B 0,C 180,E1 -8484.737,E2 -8484.737} C_VEL
LIN {X 0,Y 453.464,Z 139.625,A -85,B 0,C 180,E1 -8487.943,E2 -8487.943} C_VEL
LIN {X 0,Y 453.475,Z 139.606,A -85,B 0,C 180,E1 -8490.76,E2 -8490.76} C_VEL
LIN {X 0,Y 453.467,Z 139.609,A -85,B 0,C 180,E1 -8493.914,E2 -8493.914} C_VEL
LIN {X 0,Y 453.45,Z 139.629,A -85,B 0,C 180,E1 -8497.19,E2 -8497.19} C_VEL
LIN {X 0,Y 453.47,Z 139.599,A -85,B 0,C 180,E1 -8500.612,E2 -8500.612} C_VEL
LIN {X 0,Y 453.458,Z 139.622,A -85,B 0,C 180,E1 -8504.222,E2 -8504.222} C_VEL
LIN {X 0,Y 453.422,Z 139.622,A -85,B 0,C 180,E1 -8507,E2 -8507} C_VEL
LIN {X 0,Y 453.471,Z 139.616,A -85,B 0,C 180,E1 -8509.413,E2 -8509.413} C_VEL
LIN {X 0,Y 453.449,Z 139.625,A -85,B 0,C 180,E1 -8512.81,E2 -8512.81} C_VEL
LIN {X 0,Y 453.467,Z 139.621,A -85,B 0,C 180,E1 -8516.086,E2 -8516.086} C_VEL
LIN {X 0,Y 453.447,Z 139.605,A -85,B 0,C 180,E1 -8519.238,E2 -8519.238} C_VEL
LIN {X 0,Y 453.474,Z 139.785,A -85,B 0,C 180,E1 -8521.032,E2 -8521.032} C_VEL
LIN {X 0,Y 455.791,Z 149.45,A -85,B 0,C 180,E1 -8522.944,E2 -8522.944} C_VEL
LIN {X 0,Y 457.958,Z 159.886,A -85,B 0,C 180,E1 -8524.883,E2 -8524.883} C_VEL
LIN {X 0,Y 457.949,Z 162.097,A -85,B 0,C 180,E1 -8525.179,E2 -8525.179} C_VEL
LIN {X 0,Y 462.987,Z 185.176,A -85,B 0,C 180,E1 -8525.863,E2 -8525.863} C_VEL
LIN {X 0,Y 461.823,Z 279.846,A -85,B 0,C 180,E1 -8527.371,E2 -8527.371} C_VEL
LIN {X 0,Y 461.059,Z 285.695,A -85,B 0,C 180,E1 -8527.428,E2 -8527.428} C_VEL
LIN {X 0,Y 455.486,Z 304.733,A -85,B 0,C 180,E1 -8527.454,E2 -8527.454} C_VEL
LIN {X 0,Y 454.816,Z 310.578,A -85,B 0,C 180,E1 -8527.517,E2 -8527.517} C_VEL
LIN {X 0,Y 454.44,Z 330.43,A -85,B 0,C 180,E1 -8527.884,E2 -8527.884} C_VEL
LIN {X 0,Y 453.841,Z 346.516,A -85,B 0,C 180,E1 -8528.376,E2 -8528.376} C_VEL
LIN {X 0,Y 453.148,Z 361.254,A -85,B 0,C 180,E1 -8529.018,E2 -8529.018} C_VEL
LIN {X 0,Y 452.26,Z 374.689,A -85,B 0,C 180,E1 -8529.772,E2 -8529.772} C_VEL
LIN {X 0,Y 451.39,Z 387.648,A -85,B 0,C 180,E1 -8530.679,E2 -8530.679} C_VEL
LIN {X 0,Y 450.387,Z 399.721,A -85,B 0,C 180,E1 -8531.697,E2 -8531.697} C_VEL
LIN {X 0,Y 449.418,Z 411.973,A -85,B 0,C 180,E1 -8532.95,E2 -8532.95} C_VEL
LIN {X 0,Y 448.469,Z 423.136,A -85,B 0,C 180,E1 -8534.316,E2 -8534.316} C_VEL
LIN {X 0,Y 447.544,Z 433.983,A -85,B 0,C 180,E1 -8535.912,E2 -8535.912} C_VEL
LIN {X 0,Y 446.835,Z 442.985,A -85,B 0,C 180,E1 -8537.51,E2 -8537.51} C_VEL
LIN {X 0,Y 446.344,Z 450.447,A -85,B 0,C 180,E1 -8539.109,E2 -8539.109} C_VEL
LIN {X 0,Y 445.897,Z 457.426,A -85,B 0,C 180,E1 -8540.932,E2 -8540.932} C_VEL
LIN {X 0,Y 445.592,Z 462.913,A -85,B 0,C 180,E1 -8542.751,E2 -8542.751} C_VEL
LIN {X 0,Y 445.482,Z 467.057,A -85,B 0,C 180,E1 -8544.568,E2 -8544.568} C_VEL
LIN {X 0,Y 445.367,Z 469.971,A -85,B 0,C 180,E1 -8546.381,E2 -8546.381} C_VEL
LIN {X 0,Y 445.353,Z 471.726,A -85,B 0,C 180,E1 -8548.191,E2 -8548.191} C_VEL
LIN {X 0,Y 445.314,Z 472.34,A -85,B 0,C 180,E1 -8550,E2 -8550} C_VEL
LIN {X 0,Y 445.354,Z 471.777,A -85,B 0,C 180,E1 -8551.809,E2 -8551.809} C_VEL
LIN {X 0,Y 445.367,Z 470.09,A -85,B 0,C 180,E1 -8553.619,E2 -8553.619} C_VEL
LIN {X 0,Y 445.468,Z 467.24,A -85,B 0,C 180,E1 -8555.432,E2 -8555.432} C_VEL
LIN {X 0,Y 445.589,Z 463.161,A -85,B 0,C 180,E1 -8557.249,E2 -8557.249} C_VEL
LIN {X 0,Y 445.882,Z 457.751,A -85,B 0,C 180,E1 -8559.069,E2 -8559.069} C_VEL
LIN {X 0,Y 446.339,Z 450.86,A -85,B 0,C 180,E1 -8560.892,E2 -8560.892} C_VEL
LIN {X 0,Y 446.783,Z 443.45,A -85,B 0,C 180,E1 -8562.491,E2 -8562.491} C_VEL
LIN {X 0,Y 447.482,Z 434.526,A -85,B 0,C 180,E1 -8564.09,E2 -8564.09} C_VEL
LIN {X 0,Y 448.257,Z 425.429,A -85,B 0,C 180,E1 -8565.458,E2 -8565.458} C_VEL
LIN {X 0,Y 449.208,Z 414.699,A -85,B 0,C 180,E1 -8566.824,E2 -8566.824} C_VEL
LIN {X 0,Y 450.141,Z 402.975,A -85,B 0,C 180,E1 -8568.079,E2 -8568.079} C_VEL
LIN {X 0,Y 451.198,Z 390.203,A -85,B 0,C 180,E1 -8569.211,E2 -8569.211} C_VEL
LIN {X 0,Y 452.065,Z 377.86,A -85,B 0,C 180,E1 -8570.119,E2 -8570.119} C_VEL
LIN {X 0,Y 452.954,Z 364.62,A -85,B 0,C 180,E1 -8570.908,E2 -8570.908} C_VEL
LIN {X 0,Y 453.691,Z 350.249,A -85,B 0,C 180,E1 -8571.578,E2 -8571.578} C_VEL
LIN {X 0,Y 454.274,Z 335.098,A -85,B 0,C 180,E1 -8572.095,E2 -8572.095} C_VEL
LIN {X 0,Y 454.748,Z 319.662,A -85,B 0,C 180,E1 -8572.429,E2 -8572.429} C_VEL
LIN {X 0,Y 456.53,Z 186.297,A -85,B 0,C 180,E1 -8574.578,E2 -8574.578} C_VEL
LIN {X 0,Y 451.215,Z 162.189,A -85,B 0,C 180,E1 -8575.315,E2 -8575.315} C_VEL
LIN {X 0,Y 450.955,Z 160.35,A -85,B 0,C 180,E1 -8575.563,E2 -8575.563} C_VEL
LIN {X 0,Y 447.593,Z 145.349,A -85,B 0,C 180,E1 -8578.442,E2 -8578.442} C_VEL
LIN {X 0,Y 446.497,Z 140.933,A -85,B 0,C 180,E1 -8579.33,E2 -8579.33} C_VEL
LIN {X 0,Y 446.429,Z 140.491,A -85,B 0,C 180,E1 -8579.584,E2 -8579.584} C_VEL
LIN {X 0,Y 446.408,Z 140.505,A -85,B 0,C 180,E1 -8582.363,E2 -8582.363} C_VEL
LIN {X 0,Y 446.422,Z 140.506,A -85,B 0,C 180,E1 -8585.052,E2 -8585.052} C_VEL
LIN {X 0,Y 446.398,Z 140.504,A -85,B 0,C 180,E1 -8588.076,E2 -8588.076} C_VEL
LIN {X 0,Y 446.401,Z 140.505,A -85,B 0,C 180,E1 -8591.394,E2 -8591.394} C_VEL
LIN {X 0,Y 446.422,Z 140.495,A -85,B 0,C 180,E1 -8595.108,E2 -8595.108} C_VEL
LIN {X 0,Y 446.401,Z 140.49,A -85,B 0,C 180,E1 -8598.606,E2 -8598.606} C_VEL
LIN {X 0,Y 446.408,Z 140.494,A -85,B 0,C 180,E1 -8601.922,E2 -8601.922} C_VEL
LIN {X 0,Y 446.423,Z 140.493,A -85,B 0,C 180,E1 -8605.476,E2 -8605.476} C_VEL
LIN {X 0,Y 446.409,Z 140.475,A -85,B 0,C 180,E1 -8608.699,E2 -8608.699} C_VEL
LIN {X 0,Y 446.425,Z 140.499,A -85,B 0,C 180,E1 -8611.836,E2 -8611.836} C_VEL
LIN {X 0,Y 446.423,Z 140.492,A -85,B 0,C 180,E1 -8614.845,E2 -8614.845} C_VEL
LIN {X 0,Y 446.45,Z 140.497,A -85,B 0,C 180,E1 -8618.245,E2 -8618.245} C_VEL
LIN {X 0,Y 446.442,Z 140.494,A -85,B 0,C 180,E1 -8621.648,E2 -8621.648} C_VEL
LIN {X 0,Y 446.462,Z 140.488,A -85,B 0,C 180,E1 -8624.478,E2 -8624.478} C_VEL
LIN {X 0,Y 446.518,Z 140.485,A -85,B 0,C 180,E1 -8627.384,E2 -8627.384} C_VEL
LIN {X 0,Y 446.533,Z 140.477,A -85,B 0,C 180,E1 -8630.944,E2 -8630.944} C_VEL
LIN {X 0,Y 446.621,Z 140.476,A -85,B 0,C 180,E1 -8633.676,E2 -8633.676} C_VEL
LIN {X 0,Y 446.664,Z 140.462,A -85,B 0,C 180,E1 -8637.294,E2 -8637.294} C_VEL
LIN {X 0,Y 446.789,Z 140.454,A -85,B 0,C 180,E1 -8640,E2 -8640} C_VEL
LIN {X 0,Y 446.684,Z 140.46,A -85,B 0,C 180,E1 -8642.705,E2 -8642.705} C_VEL
LIN {X 0,Y 446.623,Z 140.473,A -85,B 0,C 180,E1 -8646.324,E2 -8646.324} C_VEL
LIN {X 0,Y 446.522,Z 140.479,A -85,B 0,C 180,E1 -8649.97,E2 -8649.97} C_VEL
LIN {X 0,Y 446.524,Z 140.488,A -85,B 0,C 180,E1 -8652.73,E2 -8652.73} C_VEL
LIN {X 0,Y 446.49,Z 140.484,A -85,B 0,C 180,E1 -8656.459,E2 -8656.459} C_VEL
LIN {X 0,Y 446.47,Z 140.492,A -85,B 0,C 180,E1 -8659.303,E2 -8659.303} C_VEL
LIN {X 0,Y 446.419,Z 140.495,A -85,B 0,C 180,E1 -8662.199,E2 -8662.199} C_VEL
LIN {X 0,Y 446.44,Z 140.492,A -85,B 0,C 180,E1 -8665.153,E2 -8665.153} C_VEL
LIN {X 0,Y 446.486,Z 140.492,A -85,B 0,C 180,E1 -8668.178,E2 -8668.178} C_VEL
LIN {X 0,Y 446.415,Z 140.484,A -85,B 0,C 180,E1 -8671.3,E2 -8671.3} C_VEL
LIN {X 0,Y 446.423,Z 140.483,A -85,B 0,C 180,E1 -8674.523,E2 -8674.523} C_VEL
LIN {X 0,Y 446.417,Z 140.503,A -85,B 0,C 180,E1 -8678.079,E2 -8678.079} C_VEL
LIN {X 0,Y 446.428,Z 140.484,A -85,B 0,C 180,E1 -8680.917,E2 -8680.917} C_VEL
LIN {X 0,Y 446.401,Z 140.505,A -85,B 0,C 180,E1 -8683.846,E2 -8683.846} C_VEL
LIN {X 0,Y 446.398,Z 140.492,A -85,B 0,C 180,E1 -8686.403,E2 -8686.403} C_VEL
LIN {X 0,Y 446.427,Z 140.498,A -85,B 0,C 180,E1 -8689.082,E2 -8689.082} C_VEL
LIN {X 0,Y 446.426,Z 140.504,A -85,B 0,C 180,E1 -8692.123,E2 -8692.123} C_VEL
LIN {X 0,Y 446.43,Z 140.502,A -85,B 0,C 180,E1 -8695.477,E2 -8695.477} C_VEL
LIN {X 0,Y 446.417,Z 140.47,A -85,B 0,C 180,E1 -8698.7,E2 -8698.7} C_VEL
LIN {X 0,Y 446.472,Z 140.667,A -85,B 0,C 180,E1 -8699.558,E2 -8699.558} C_VEL
LIN {X 0,Y 449.956,Z 154.899,A -85,B 0,C 180,E1 -8702.271,E2 -8702.271} C_VEL
LIN {X 0,Y 451.428,Z 162.6,A -85,B 0,C 180,E1 -8703.66,E2 -8703.66} C_VEL
LIN {X 0,Y 451.029,Z 169.215,A -85,B 0,C 180,E1 -8704.698,E2 -8704.698} C_VEL
LIN {X 0,Y 456.393,Z 195.053,A -85,B 0,C 180,E1 -8705.476,E2 -8705.476} C_VEL
LIN {X 0,Y 454.91,Z 306.954,A -85,B 0,C 180,E1 -8707.28,E2 -8707.28} C_VEL
LIN {X 0,Y 454.439,Z 336.75,A -85,B 0,C 180,E1 -8707.794,E2 -8707.794} C_VEL
LIN {X 0,Y 453.831,Z 352.054,A -85,B 0,C 180,E1 -8708.235,E2 -8708.235} C_VEL
LIN {X 0,Y 453.169,Z 366.337,A -85,B 0,C 180,E1 -8708.821,E2 -8708.821} C_VEL
LIN {X 0,Y 452.335,Z 379.779,A -85,B 0,C 180,E1 -8709.538,E2 -8709.538} C_VEL
LIN {X 0,Y 451.337,Z 393.256,A -85,B 0,C 180,E1 -8710.44,E2 -8710.44} C_VEL
LIN {X 0,Y 450.293,Z 406.973,A -85,B 0,C 180,E1 -8711.575,E2 -8711.575} C_VEL
LIN {X 0,Y 449.254,Z 419.387,A -85,B 0,C 180,E1 -8712.826,E2 -8712.826} C_VEL
LIN {X 0,Y 448.216,Z 431.557,A -85,B 0,C 180,E1 -8714.307,E2 -8714.307} C_VEL
LIN {X 0,Y 447.351,Z 442.375,A -85,B 0,C 180,E1 -8715.906,E2 -8715.906} C_VEL
LIN {X 0,Y 446.671,Z 451.166,A -85,B 0,C 180,E1 -8717.462,E2 -8717.462} C_VEL
LIN {X 0,Y 446.26,Z 458.854,A -85,B 0,C 180,E1 -8719.106,E2 -8719.106} C_VEL
LIN {X 0,Y 445.797,Z 465.822,A -85,B 0,C 180,E1 -8720.929,E2 -8720.929} C_VEL
LIN {X 0,Y 445.578,Z 471.3,A -85,B 0,C 180,E1 -8722.751,E2 -8722.751} C_VEL
LIN {X 0,Y 445.439,Z 475.441,A -85,B 0,C 180,E1 -8724.568,E2 -8724.568} C_VEL
LIN {X 0,Y 445.324,Z 478.342,A -85,B 0,C 180,E1 -8726.381,E2 -8726.381} C_VEL
LIN {X 0,Y 445.348,Z 480.073,A -85,B 0,C 180,E1 -8728.191,E2 -8728.191} C_VEL
LIN {X 0,Y 445.313,Z 480.666,A -85,B 0,C 180,E1 -8730,E2 -8730} C_VEL
LIN {X 0,Y 445.348,Z 480.07,A -85,B 0,C 180,E1 -8731.809,E2 -8731.809} C_VEL
LIN {X 0,Y 445.325,Z 478.334,A -85,B 0,C 180,E1 -8733.619,E2 -8733.619} C_VEL
LIN {X 0,Y 445.449,Z 475.434,A -85,B 0,C 180,E1 -8735.432,E2 -8735.432} C_VEL
LIN {X 0,Y 445.579,Z 471.297,A -85,B 0,C 180,E1 -8737.249,E2 -8737.249} C_VEL
LIN {X 0,Y 445.797,Z 465.814,A -85,B 0,C 180,E1 -8739.071,E2 -8739.071} C_VEL
LIN {X 0,Y 446.262,Z 458.836,A -85,B 0,C 180,E1 -8740.893,E2 -8740.893} C_VEL
LIN {X 0,Y 446.642,Z 451.239,A -85,B 0,C 180,E1 -8742.52,E2 -8742.52} C_VEL
LIN {X 0,Y 447.351,Z 442.358,A -85,B 0,C 180,E1 -8744.094,E2 -8744.094} C_VEL
LIN {X 0,Y 448.226,Z 431.532,A -85,B 0,C 180,E1 -8745.692,E2 -8745.692} C_VEL
LIN {X 0,Y 449.214,Z 419.36,A -85,B 0,C 180,E1 -8747.176,E2 -8747.176} C_VEL
LIN {X 0,Y 450.297,Z 406.943,A -85,B 0,C 180,E1 -8748.424,E2 -8748.424} C_VEL
LIN {X 0,Y 451.232,Z 394.721,A -85,B 0,C 180,E1 -8749.446,E2 -8749.446} C_VEL
LIN {X 0,Y 452.179,Z 381.521,A -85,B 0,C 180,E1 -8750.351,E2 -8750.351} C_VEL
LIN {X 0,Y 453.078,Z 367.548,A -85,B 0,C 180,E1 -8751.115,E2 -8751.115} C_VEL
LIN {X 0,Y 453.766,Z 353.516,A -85,B 0,C 180,E1 -8751.708,E2 -8751.708} C_VEL
LIN {X 0,Y 454.35,Z 338.874,A -85,B 0,C 180,E1 -8752.15,E2 -8752.15} C_VEL
LIN {X 0,Y 454.748,Z 319.215,A -85,B 0,C 180,E1 -8752.519,E2 -8752.519} C_VEL
LIN {X 0,Y 456.447,Z 195.875,A -85,B 0,C 180,E1 -8754.502,E2 -8754.502} C_VEL
LIN {X 0,Y 451.03,Z 169.481,A -85,B 0,C 180,E1 -8755.28,E2 -8755.28} C_VEL
LIN {X 0,Y 451.132,Z 166.616,A -85,B 0,C 180,E1 -8755.684,E2 -8755.684} C_VEL
LIN {X 0,Y 451.288,Z 161.075,A -85,B 0,C 180,E1 -8756.598,E2 -8756.598} C_VEL
LIN {X 0,Y 448.215,Z 147.623,A -85,B 0,C 180,E1 -8759.083,E2 -8759.083} C_VEL
LIN {X 0,Y 446.467,Z 140.585,A -85,B 0,C 180,E1 -8760.475,E2 -8760.475} C_VEL
LIN {X 0,Y 446.445,Z 140.489,A -85,B 0,C 180,E1 -8763.454,E2 -8763.454} C_VEL
LIN {X 0,Y 446.402,Z 140.502,A -85,B 0,C 180,E1 -8766.745,E2 -8766.745} C_VEL
LIN {X 0,Y 446.45,Z 140.487,A -85,B 0,C 180,E1 -8769.524,E2 -8769.524} C_VEL
LIN {X 0,Y 446.429,Z 140.495,A -85,B 0,C 180,E1 -8772.605,E2 -8772.605} C_VEL
LIN {X 0,Y 446.452,Z 140.49,A -85,B 0,C 180,E1 -8775.104,E2 -8775.104} C_VEL
LIN {X 0,Y 446.428,Z 140.487,A -85,B 0,C 180,E1 -8778.609,E2 -8778.609} C_VEL
LIN {X 0,Y 446.444,Z 140.487,A -85,B 0,C 180,E1 -8780.973,E2 -8780.973} C_VEL
LIN {X 0,Y 446.418,Z 140.495,A -85,B 0,C 180,E1 -8784.374,E2 -8784.374} C_VEL
LIN {X 0,Y 446.417,Z 140.474,A -85,B 0,C 180,E1 -8787.638,E2 -8787.638} C_VEL
LIN {X 0,Y 446.449,Z 140.495,A -85,B 0,C 180,E1 -8790.791,E2 -8790.791} C_VEL
LIN {X 0,Y 446.479,Z 140.486,A -85,B 0,C 180,E1 -8793.849,E2 -8793.849} C_VEL
LIN {X 0,Y 446.43,Z 140.501,A -85,B 0,C 180,E1 -8796.823,E2 -8796.823} C_VEL
LIN {X 0,Y 446.444,Z 140.493,A -85,B 0,C 180,E1 -8799.737,E2 -8799.737} C_VEL
LIN {X 0,Y 446.456,Z 140.497,A -85,B 0,C 180,E1 -8802.597,E2 -8802.597} C_VEL
LIN {X 0,Y 446.47,Z 140.492,A -85,B 0,C 180,E1 -8805.412,E2 -8805.412} C_VEL
LIN {X 0,Y 446.519,Z 140.487,A -85,B 0,C 180,E1 -8808.193,E2 -8808.193} C_VEL
LIN {X 0,Y 446.534,Z 140.48,A -85,B 0,C 180,E1 -8810.945,E2 -8810.945} C_VEL
LIN {X 0,Y 446.622,Z 140.472,A -85,B 0,C 180,E1 -8813.676,E2 -8813.676} C_VEL
LIN {X 0,Y 446.684,Z 140.46,A -85,B 0,C 180,E1 -8817.295,E2 -8817.295} C_VEL
LIN {X 0,Y 446.791,Z 140.453,A -85,B 0,C 180,E1 -8820,E2 -8820} C_VEL
LIN {X 0,Y 446.679,Z 140.46,A -85,B 0,C 180,E1 -8822.706,E2 -8822.706} C_VEL
LIN {X 0,Y 446.621,Z 140.477,A -85,B 0,C 180,E1 -8826.324,E2 -8826.324} C_VEL
LIN {X 0,Y 446.522,Z 140.483,A -85,B 0,C 180,E1 -8829.97,E2 -8829.97} C_VEL
LIN {X 0,Y 446.523,Z 140.484,A -85,B 0,C 180,E1 -8832.73,E2 -8832.73} C_VEL
LIN {X 0,Y 446.484,Z 140.493,A -85,B 0,C 180,E1 -8836.459,E2 -8836.459} C_VEL
LIN {X 0,Y 446.469,Z 140.489,A -85,B 0,C 180,E1 -8839.303,E2 -8839.303} C_VEL
LIN {X 0,Y 446.419,Z 140.502,A -85,B 0,C 180,E1 -8842.2,E2 -8842.2} C_VEL
LIN {X 0,Y 446.422,Z 140.492,A -85,B 0,C 180,E1 -8845.155,E2 -8845.155} C_VEL
LIN {X 0,Y 446.437,Z 140.498,A -85,B 0,C 180,E1 -8848.182,E2 -8848.182} C_VEL
LIN {X 0,Y 446.413,Z 140.476,A -85,B 0,C 180,E1 -8851.301,E2 -8851.301} C_VEL
LIN {X 0,Y 446.423,Z 140.493,A -85,B 0,C 180,E1 -8854.524,E2 -8854.524} C_VEL
LIN {X 0,Y 446.411,Z 140.494,A -85,B 0,C 180,E1 -8858.078,E2 -8858.078} C_VEL
LIN {X 0,Y 446.401,Z 140.487,A -85,B 0,C 180,E1 -8861.394,E2 -8861.394} C_VEL
LIN {X 0,Y 446.45,Z 140.49,A -85,B 0,C 180,E1 -8865.104,E2 -8865.104} C_VEL
LIN {X 0,Y 446.401,Z 140.505,A -85,B 0,C 180,E1 -8868.606,E2 -8868.606} C_VEL
LIN {X 0,Y 446.41,Z 140.503,A -85,B 0,C 180,E1 -8871.922,E2 -8871.922} C_VEL
LIN {X 0,Y 446.422,Z 140.501,A -85,B 0,C 180,E1 -8875.476,E2 -8875.476} C_VEL
LIN {X 0,Y 446.392,Z 140.491,A -85,B 0,C 180,E1 -8878.698,E2 -8878.698} C_VEL
LIN {X 0,Y 446.439,Z 140.627,A -85,B 0,C 180,E1 -8880.666,E2 -8880.666} C_VEL
LIN {X 0,Y 448.904,Z 150.937,A -85,B 0,C 180,E1 -8882.746,E2 -8882.746} C_VEL
LIN {X 0,Y 451.188,Z 161.694,A -85,B 0,C 180,E1 -8884.75,E2 -8884.75} C_VEL
LIN {X 0,Y 454.06,Z 174.862,A -85,B 0,C 180,E1 -8885.179,E2 -8885.179} C_VEL
LIN {X 0,Y 456.544,Z 186.686,A -85,B 0,C 180,E1 -8885.524,E2 -8885.524} C_VEL
LIN {X 0,Y 454.816,Z 310.578,A -85,B 0,C 180,E1 -8887.517,E2 -8887.517} C_VEL
LIN {X 0,Y 454.096,Z 316.427,A -85,B 0,C 180,E1 -8887.576,E2 -8887.576} C_VEL
LIN {X 0,Y 448.71,Z 333.456,A -85,B 0,C 180,E1 -8887.665,E2 -8887.665} C_VEL
LIN {X 0,Y 447.621,Z 339.182,A -85,B 0,C 180,E1 -8887.787,E2 -8887.787} C_VEL
LIN {X 0,Y 447.511,Z 341.096,A -85,B 0,C 180,E1 -8887.845,E2 -8887.845} C_VEL
LIN {X 0,Y 446.878,Z 355.149,A -85,B 0,C 180,E1 -8888.396,E2 -8888.396} C_VEL
LIN {X 0,Y 446.01,Z 369.12,A -85,B 0,C 180,E1 -8889.114,E2 -8889.114} C_VEL
LIN {X 0,Y 444.961,Z 383.14,A -85,B 0,C 180,E1 -8890.028,E2 -8890.028} C_VEL
LIN {X 0,Y 443.937,Z 395.955,A -85,B 0,C 180,E1 -8891.062,E2 -8891.062} C_VEL
LIN {X 0,Y 442.979,Z 407.293,A -85,B 0,C 180,E1 -8892.161,E2 -8892.161} C_VEL
LIN {X 0,Y 441.998,Z 417.872,A -85,B 0,C 180,E1 -8893.369,E2 -8893.369} C_VEL
LIN {X 0,Y 441.124,Z 428.095,A -85,B 0,C 180,E1 -8894.759,E2 -8894.759} C_VEL
LIN {X 0,Y 440.256,Z 438.237,A -85,B 0,C 180,E1 -8896.405,E2 -8896.405} C_VEL
LIN {X 0,Y 439.609,Z 447.499,A -85,B 0,C 180,E1 -8898.239,E2 -8898.239} C_VEL
LIN {X 0,Y 439.026,Z 454.204,A -85,B 0,C 180,E1 -8899.858,E2 -8899.858} C_VEL
LIN {X 0,Y 438.69,Z 460.414,A -85,B 0,C 180,E1 -8901.71,E2 -8901.71} C_VEL
LIN {X 0,Y 438.47,Z 465.308,A -85,B 0,C 180,E1 -8903.6,E2 -8903.6} C_VEL
LIN {X 0,Y 438.314,Z 468.729,A -85,B 0,C 180,E1 -8905.402,E2 -8905.402} C_VEL
LIN {X 0,Y 438.335,Z 471.056,A -85,B 0,C 180,E1 -8907.243,E2 -8907.243} C_VEL
LIN {X 0,Y 438.228,Z 472.248,A -85,B 0,C 180,E1 -8909.081,E2 -8909.081} C_VEL
LIN {X 0,Y 438.228,Z 472.265,A -85,B 0,C 180,E1 -8910.919,E2 -8910.919} C_VEL
LIN {X 0,Y 438.335,Z 471.141,A -85,B 0,C 180,E1 -8912.757,E2 -8912.757} C_VEL
LIN {X 0,Y 438.311,Z 468.88,A -85,B 0,C 180,E1 -8914.598,E2 -8914.598} C_VEL
LIN {X 0,Y 438.422,Z 465.425,A -85,B 0,C 180,E1 -8916.443,E2 -8916.443} C_VEL
LIN {X 0,Y 438.654,Z 460.695,A -85,B 0,C 180,E1 -8918.291,E2 -8918.291} C_VEL
LIN {X 0,Y 439,Z 454.569,A -85,B 0,C 180,E1 -8920.143,E2 -8920.143} C_VEL
LIN {X 0,Y 439.564,Z 447.91,A -85,B 0,C 180,E1 -8921.763,E2 -8921.763} C_VEL
LIN {X 0,Y 440.095,Z 440.114,A -85,B 0,C 180,E1 -8923.342,E2 -8923.342} C_VEL
LIN {X 0,Y 440.94,Z 430.221,A -85,B 0,C 180,E1 -8925.011,E2 -8925.011} C_VEL
LIN {X 0,Y 441.788,Z 420.359,A -85,B 0,C 180,E1 -8926.402,E2 -8926.402} C_VEL
LIN {X 0,Y 442.815,Z 408.78,A -85,B 0,C 180,E1 -8927.773,E2 -8927.773} C_VEL
LIN {X 0,Y 443.97,Z 395.675,A -85,B 0,C 180,E1 -8929.056,E2 -8929.056} C_VEL
LIN {X 0,Y 445.015,Z 382.808,A -85,B 0,C 180,E1 -8930.09,E2 -8930.09} C_VEL
LIN {X 0,Y 446.048,Z 368.698,A -85,B 0,C 180,E1 -8931.005,E2 -8931.005} C_VEL
LIN {X 0,Y 446.931,Z 353.657,A -85,B 0,C 180,E1 -8931.766,E2 -8931.766} C_VEL
LIN {X 0,Y 447.61,Z 338.82,A -85,B 0,C 180,E1 -8932.32,E2 -8932.32} C_VEL
LIN {X 0,Y 448.073,Z 324.226,A -85,B 0,C 180,E1 -8932.69,E2 -8932.69} C_VEL
LIN {X 0,Y 450.14,Z 188.567,A -85,B 0,C 180,E1 -8934.912,E2 -8934.912} C_VEL
LIN {X 0,Y 445.432,Z 166.099,A -85,B 0,C 180,E1 -8935.587,E2 -8935.587} C_VEL
LIN {X 0,Y 444.055,Z 161.66,A -85,B 0,C 180,E1 -8935.791,E2 -8935.791} C_VEL
LIN {X 0,Y 440.807,Z 147.296,A -85,B 0,C 180,E1 -8938.575,E2 -8938.575} C_VEL
LIN {X 0,Y 439.434,Z 141.725,A -85,B 0,C 180,E1 -8939.722,E2 -8939.722} C_VEL
LIN {X 0,Y 439.366,Z 141.355,A -85,B 0,C 180,E1 -8940.092,E2 -8940.092} C_VEL
LIN {X 0,Y 439.367,Z 141.38,A -85,B 0,C 180,E1 -8942.947,E2 -8942.947} C_VEL
LIN {X 0,Y 439.366,Z 141.373,A -85,B 0,C 180,E1 -8946.288,E2 -8946.288} C_VEL
LIN {X 0,Y 439.359,Z 141.369,A -85,B 0,C 180,E1 -8949.78,E2 -8949.78} C_VEL
LIN {X 0,Y 439.333,Z 141.385,A -85,B 0,C 180,E1 -8952.62,E2 -8952.62} C_VEL
LIN {X 0,Y 439.376,Z 141.375,A -85,B 0,C 180,E1 -8955.267,E2 -8955.267} C_VEL
LIN {X 0,Y 439.363,Z 141.363,A -85,B 0,C 180,E1 -8958.747,E2 -8958.747} C_VEL
LIN {X 0,Y 439.363,Z 141.37,A -85,B 0,C 180,E1 -8961.61,E2 -8961.61} C_VEL
LIN {X 0,Y 439.396,Z 141.372,A -85,B 0,C 180,E1 -8964.844,E2 -8964.844} C_VEL
LIN {X 0,Y 439.367,Z 141.346,A -85,B 0,C 180,E1 -8968.139,E2 -8968.139} C_VEL
LIN {X 0,Y 439.401,Z 141.372,A -85,B 0,C 180,E1 -8971.606,E2 -8971.606} C_VEL
LIN {X 0,Y 439.367,Z 141.373,A -85,B 0,C 180,E1 -8974.413,E2 -8974.413} C_VEL
LIN {X 0,Y 439.365,Z 141.378,A -85,B 0,C 180,E1 -8977.424,E2 -8977.424} C_VEL
LIN {X 0,Y 439.443,Z 141.365,A -85,B 0,C 180,E1 -8980.663,E2 -8980.663} C_VEL
LIN {X 0,Y 439.421,Z 141.368,A -85,B 0,C 180,E1 -8984.223,E2 -8984.223} C_VEL
LIN {X 0,Y 439.487,Z 141.36,A -85,B 0,C 180,E1 -8987.285,E2 -8987.285} C_VEL
LIN {X 0,Y 439.496,Z 141.354,A -85,B 0,C 180,E1 -8990.798,E2 -8990.798} C_VEL
LIN {X 0,Y 439.593,Z 141.35,A -85,B 0,C 180,E1 -8993.574,E2 -8993.574} C_VEL
LIN {X 0,Y 439.616,Z 141.339,A -85,B 0,C 180,E1 -8997.251,E2 -8997.251} C_VEL
LIN {X 0,Y 439.759,Z 141.33,A -85,B 0,C 180,E1 -9000,E2 -9000} C_VEL
LIN {X 0,Y 439.633,Z 141.338,A -85,B 0,C 180,E1 -9002.749,E2 -9002.749} C_VEL
LIN {X 0,Y 439.594,Z 141.348,A -85,B 0,C 180,E1 -9006.425,E2 -9006.425} C_VEL
LIN {X 0,Y 439.497,Z 141.355,A -85,B 0,C 180,E1 -9009.202,E2 -9009.202} C_VEL
LIN {X 0,Y 439.467,Z 141.37,A -85,B 0,C 180,E1 -9012.937,E2 -9012.937} C_VEL
LIN {X 0,Y 439.448,Z 141.36,A -85,B 0,C 180,E1 -9016.348,E2 -9016.348} C_VEL
LIN {X 0,Y 439.403,Z 141.37,A -85,B 0,C 180,E1 -9019.626,E2 -9019.626} C_VEL
LIN {X 0,Y 439.365,Z 141.377,A -85,B 0,C 180,E1 -9022.575,E2 -9022.575} C_VEL
LIN {X 0,Y 439.388,Z 141.367,A -85,B 0,C 180,E1 -9025.586,E2 -9025.586} C_VEL
LIN {X 0,Y 439.418,Z 141.378,A -85,B 0,C 180,E1 -9028.673,E2 -9028.673} C_VEL
LIN {X 0,Y 439.366,Z 141.354,A -85,B 0,C 180,E1 -9032.029,E2 -9032.029} C_VEL
LIN {X 0,Y 439.393,Z 141.371,A -85,B 0,C 180,E1 -9035.34,E2 -9035.34} C_VEL
LIN {X 0,Y 439.379,Z 141.37,A -85,B 0,C 180,E1 -9038.595,E2 -9038.595} C_VEL
LIN {X 0,Y 439.389,Z 141.363,A -85,B 0,C 180,E1 -9041.257,E2 -9041.257} C_VEL
LIN {X 0,Y 439.4,Z 141.368,A -85,B 0,C 180,E1 -9044.729,E2 -9044.729} C_VEL
LIN {X 0,Y 439.397,Z 141.374,A -85,B 0,C 180,E1 -9047.796,E2 -9047.796} C_VEL
LIN {X 0,Y 439.395,Z 141.366,A -85,B 0,C 180,E1 -9050.224,E2 -9050.224} C_VEL
LIN {X 0,Y 439.374,Z 141.373,A -85,B 0,C 180,E1 -9053.713,E2 -9053.713} C_VEL
LIN {X 0,Y 439.372,Z 141.355,A -85,B 0,C 180,E1 -9057.054,E2 -9057.054} C_VEL
LIN {X 0,Y 439.44,Z 141.542,A -85,B 0,C 180,E1 -9059.184,E2 -9059.184} C_VEL
LIN {X 0,Y 442.792,Z 155.066,A -85,B 0,C 180,E1 -9061.823,E2 -9061.823} C_VEL
LIN {X 0,Y 444.616,Z 164.026,A -85,B 0,C 180,E1 -9063.478,E2 -9063.478} C_VEL
LIN {X 0,Y 444.326,Z 169.28,A -85,B 0,C 180,E1 -9064.296,E2 -9064.296} C_VEL
LIN {X 0,Y 449.85,Z 195.778,A -85,B 0,C 180,E1 -9065.109,E2 -9065.109} C_VEL
LIN {X 0,Y 449.314,Z 247.434,A -85,B 0,C 180,E1 -9065.965,E2 -9065.965} C_VEL
LIN {X 0,Y 447.94,Z 335.556,A -85,B 0,C 180,E1 -9067.424,E2 -9067.424} C_VEL
LIN {X 0,Y 447.286,Z 351.398,A -85,B 0,C 180,E1 -9067.876,E2 -9067.876} C_VEL
LIN {X 0,Y 446.578,Z 365.619,A -85,B 0,C 180,E1 -9068.459,E2 -9068.459} C_VEL
LIN {X 0,Y 445.669,Z 379.718,A -85,B 0,C 180,E1 -9069.218,E2 -9069.218} C_VEL
LIN {X 0,Y 444.594,Z 393.193,A -85,B 0,C 180,E1 -9070.131,E2 -9070.131} C_VEL
LIN {X 0,Y 443.497,Z 406.909,A -85,B 0,C 180,E1 -9071.283,E2 -9071.283} C_VEL
LIN {X 0,Y 442.46,Z 418.981,A -85,B 0,C 180,E1 -9072.516,E2 -9072.516} C_VEL
LIN {X 0,Y 441.457,Z 429.727,A -85,B 0,C 180,E1 -9073.823,E2 -9073.823} C_VEL
LIN {X 0,Y 440.654,Z 439.385,A -85,B 0,C 180,E1 -9075.215,E2 -9075.215} C_VEL
LIN {X 0,Y 439.827,Z 448.868,A -85,B 0,C 180,E1 -9076.838,E2 -9076.838} C_VEL
LIN {X 0,Y 439.386,Z 456.769,A -85,B 0,C 180,E1 -9078.467,E2 -9078.467} C_VEL
LIN {X 0,Y 438.804,Z 464.141,A -85,B 0,C 180,E1 -9080.318,E2 -9080.318} C_VEL
LIN {X 0,Y 438.523,Z 469.989,A -85,B 0,C 180,E1 -9082.17,E2 -9082.17} C_VEL
LIN {X 0,Y 438.417,Z 473.7,A -85,B 0,C 180,E1 -9083.659,E2 -9083.659} C_VEL
LIN {X 0,Y 438.289,Z 476.975,A -85,B 0,C 180,E1 -9085.401,E2 -9085.401} C_VEL
LIN {X 0,Y 438.283,Z 479.285,A -85,B 0,C 180,E1 -9087.243,E2 -9087.243} C_VEL
LIN {X 0,Y 438.227,Z 480.447,A -85,B 0,C 180,E1 -9089.081,E2 -9089.081} C_VEL
LIN {X 0,Y 438.227,Z 480.446,A -85,B 0,C 180,E1 -9090.919,E2 -9090.919} C_VEL
LIN {X 0,Y 438.283,Z 479.279,A -85,B 0,C 180,E1 -9092.757,E2 -9092.757} C_VEL
LIN {X 0,Y 438.291,Z 476.966,A -85,B 0,C 180,E1 -9094.599,E2 -9094.599} C_VEL
LIN {X 0,Y 438.445,Z 473.459,A -85,B 0,C 180,E1 -9096.442,E2 -9096.442} C_VEL
LIN {X 0,Y 438.589,Z 468.665,A -85,B 0,C 180,E1 -9098.292,E2 -9098.292} C_VEL
LIN {X 0,Y 438.87,Z 462.454,A -85,B 0,C 180,E1 -9100.146,E2 -9100.146} C_VEL
LIN {X 0,Y 439.432,Z 455.737,A -85,B 0,C 180,E1 -9101.766,E2 -9101.766} C_VEL
LIN {X 0,Y 439.958,Z 447.614,A -85,B 0,C 180,E1 -9103.393,E2 -9103.393} C_VEL
LIN {X 0,Y 440.782,Z 437.874,A -85,B 0,C 180,E1 -9105.016,E2 -9105.016} C_VEL
LIN {X 0,Y 441.628,Z 427.912,A -85,B 0,C 180,E1 -9106.408,E2 -9106.408} C_VEL
LIN {X 0,Y 442.66,Z 416.296,A -85,B 0,C 180,E1 -9107.772,E2 -9107.772} C_VEL
LIN {X 0,Y 443.693,Z 404.286,A -85,B 0,C 180,E1 -9108.948,E2 -9108.948} C_VEL
LIN {X 0,Y 444.72,Z 391.546,A -85,B 0,C 180,E1 -9109.983,E2 -9109.983} C_VEL
LIN {X 0,Y 445.81,Z 377.646,A -85,B 0,C 180,E1 -9110.896,E2 -9110.896} C_VEL
LIN {X 0,Y 446.697,Z 363.14,A -85,B 0,C 180,E1 -9111.648,E2 -9111.648} C_VEL
LIN {X 0,Y 447.376,Z 349.651,A -85,B 0,C 180,E1 -9112.18,E2 -9112.18} C_VEL
LIN {X 0,Y 447.937,Z 333.998,A -85,B 0,C 180,E1 -9112.606,E2 -9112.606} C_VEL
LIN {X 0,Y 449.991,Z 197.03,A -85,B 0,C 180,E1 -9114.856,E2 -9114.856} C_VEL
LIN {X 0,Y 444.583,Z 170.748,A -85,B 0,C 180,E1 -9115.638,E2 -9115.638} C_VEL
LIN {X 0,Y 444.281,Z 168.744,A -85,B 0,C 180,E1 -9115.752,E2 -9115.752} C_VEL
LIN {X 0,Y 444.565,Z 163.989,A -85,B 0,C 180,E1 -9116.526,E2 -9116.526} C_VEL
LIN {X 0,Y 442.788,Z 155.029,A -85,B 0,C 180,E1 -9118.177,E2 -9118.177} C_VEL
LIN {X 0,Y 439.423,Z 141.46,A -85,B 0,C 180,E1 -9120.85,E2 -9120.85} C_VEL
LIN {X 0,Y 439.388,Z 141.377,A -85,B 0,C 180,E1 -9124.044,E2 -9124.044} C_VEL
LIN {X 0,Y 439.351,Z 141.381,A -85,B 0,C 180,E1 -9126.888,E2 -9126.888} C_VEL
LIN {X 0,Y 439.402,Z 141.366,A -85,B 0,C 180,E1 -9129.849,E2 -9129.849} C_VEL
LIN {X 0,Y 439.382,Z 141.373,A -85,B 0,C 180,E1 -9132.627,E2 -9132.627} C_VEL
LIN {X 0,Y 439.4,Z 141.369,A -85,B 0,C 180,E1 -9135.271,E2 -9135.271} C_VEL
LIN {X 0,Y 439.389,Z 141.362,A -85,B 0,C 180,E1 -9138.743,E2 -9138.743} C_VEL
LIN {X 0,Y 439.375,Z 141.374,A -85,B 0,C 180,E1 -9141.608,E2 -9141.608} C_VEL
LIN {X 0,Y 439.397,Z 141.369,A -85,B 0,C 180,E1 -9144.844,E2 -9144.844} C_VEL
LIN {X 0,Y 439.37,Z 141.358,A -85,B 0,C 180,E1 -9148.139,E2 -9148.139} C_VEL
LIN {X 0,Y 439.433,Z 141.372,A -85,B 0,C 180,E1 -9151.598,E2 -9151.598} C_VEL
LIN {X 0,Y 439.401,Z 141.366,A -85,B 0,C 180,E1 -9154.415,E2 -9154.415} C_VEL
LIN {X 0,Y 439.366,Z 141.376,A -85,B 0,C 180,E1 -9157.425,E2 -9157.425} C_VEL
LIN {X 0,Y 439.442,Z 141.367,A -85,B 0,C 180,E1 -9160.663,E2 -9160.663} C_VEL
LIN {X 0,Y 439.463,Z 141.358,A -85,B 0,C 180,E1 -9164.225,E2 -9164.225} C_VEL
LIN {X 0,Y 439.485,Z 141.363,A -85,B 0,C 180,E1 -9168.001,E2 -9168.001} C_VEL
LIN {X 0,Y 439.505,Z 141.356,A -85,B 0,C 180,E1 -9171.726,E2 -9171.726} C_VEL
LIN {X 0,Y 439.612,Z 141.349,A -85,B 0,C 180,E1 -9174.496,E2 -9174.496} C_VEL
LIN {X 0,Y 439.635,Z 141.341,A -85,B 0,C 180,E1 -9178.168,E2 -9178.168} C_VEL
LIN {X 0,Y 439.76,Z 141.329,A -85,B 0,C 180,E1 -9180,E2 -9180} C_VEL
LIN {X 0,Y 439.628,Z 141.337,A -85,B 0,C 180,E1 -9182.749,E2 -9182.749} C_VEL
LIN {X 0,Y 439.593,Z 141.351,A -85,B 0,C 180,E1 -9186.426,E2 -9186.426} C_VEL
LIN {X 0,Y 439.497,Z 141.353,A -85,B 0,C 180,E1 -9189.202,E2 -9189.202} C_VEL
LIN {X 0,Y 439.467,Z 141.362,A -85,B 0,C 180,E1 -9192.938,E2 -9192.938} C_VEL
LIN {X 0,Y 439.444,Z 141.371,A -85,B 0,C 180,E1 -9196.346,E2 -9196.346} C_VEL
LIN {X 0,Y 439.403,Z 141.368,A -85,B 0,C 180,E1 -9199.626,E2 -9199.626} C_VEL
LIN {X 0,Y 439.365,Z 141.378,A -85,B 0,C 180,E1 -9202.576,E2 -9202.576} C_VEL
LIN {X 0,Y 439.367,Z 141.372,A -85,B 0,C 180,E1 -9205.587,E2 -9205.587} C_VEL
LIN {X 0,Y 439.391,Z 141.373,A -85,B 0,C 180,E1 -9208.675,E2 -9208.675} C_VEL
LIN {X 0,Y 439.363,Z 141.346,A -85,B 0,C 180,E1 -9212.029,E2 -9212.029} C_VEL
LIN {X 0,Y 439.391,Z 141.374,A -85,B 0,C 180,E1 -9215.34,E2 -9215.34} C_VEL
LIN {X 0,Y 439.362,Z 141.371,A -85,B 0,C 180,E1 -9218.597,E2 -9218.597} C_VEL
LIN {X 0,Y 439.349,Z 141.377,A -85,B 0,C 180,E1 -9222.21,E2 -9222.21} C_VEL
LIN {X 0,Y 439.397,Z 141.366,A -85,B 0,C 180,E1 -9225.27,E2 -9225.27} C_VEL
LIN {X 0,Y 439.354,Z 141.38,A -85,B 0,C 180,E1 -9229.016,E2 -9229.016} C_VEL
LIN {X 0,Y 439.345,Z 141.385,A -85,B 0,C 180,E1 -9232.564,E2 -9232.564} C_VEL
LIN {X 0,Y 439.395,Z 141.378,A -85,B 0,C 180,E1 -9234.844,E2 -9234.844} C_VEL
LIN {X 0,Y 439.356,Z 141.38,A -85,B 0,C 180,E1 -9238.138,E2 -9238.138} C_VEL
LIN {X 0,Y 439.382,Z 141.45,A -85,B 0,C 180,E1 -9240.274,E2 -9240.274} C_VEL
LIN {X 0,Y 439.951,Z 143.928,A -85,B 0,C 180,E1 -9240.842,E2 -9240.842} C_VEL
LIN {X 0,Y 442.597,Z 154.964,A -85,B 0,C 180,E1 -9243.038,E2 -9243.038} C_VEL
LIN {X 0,Y 444.138,Z 161.877,A -85,B 0,C 180,E1 -9244.331,E2 -9244.331} C_VEL
LIN {X 0,Y 445.508,Z 166.526,A -85,B 0,C 180,E1 -9244.521,E2 -9244.521} C_VEL
LIN {X 0,Y 449.993,Z 187.163,A -85,B 0,C 180,E1 -9245.151,E2 -9245.151} C_VEL
LIN {X 0,Y 448.589,Z 290.888,A -85,B 0,C 180,E1 -9246.85,E2 -9246.85} C_VEL
LIN {X 0,Y 447.996,Z 328.232,A -85,B 0,C 180,E1 -9247.488,E2 -9247.488} C_VEL
LIN {X 0,Y 447.511,Z 341.096,A -85,B 0,C 180,E1 -9247.845,E2 -9247.845} C_VEL
LIN {X 0,Y 446.694,Z 346.81,A -85,B 0,C 180,E1 -9248.012,E2 -9248.012} C_VEL
LIN {X 0,Y 443.514,Z 356.024,A -85,B 0,C 180,E1 -9248.261,E2 -9248.261} C_VEL
LIN {X 0,Y 440.26,Z 365.126,A -85,B 0,C 180,E1 -9248.578,E2 -9248.578} C_VEL
LIN {X 0,Y 439.296,Z 370.475,A -85,B 0,C 180,E1 -9248.859,E2 -9248.859} C_VEL
LIN {X 0,Y 438.167,Z 384.793,A -85,B 0,C 180,E1 -9249.827,E2 -9249.827} C_VEL
LIN {X 0,Y 437.106,Z 397.316,A -85,B 0,C 180,E1 -9250.877,E2 -9250.877} C_VEL
LIN {X 0,Y 436.111,Z 408.081,A -85,B 0,C 180,E1 -9251.952,E2 -9251.952} C_VEL
LIN {X 0,Y 434.993,Z 419.725,A -85,B 0,C 180,E1 -9253.335,E2 -9253.335} C_VEL
LIN {X 0,Y 434.086,Z 429.701,A -85,B 0,C 180,E1 -9254.746,E2 -9254.746} C_VEL
LIN {X 0,Y 433.204,Z 439.446,A -85,B 0,C 180,E1 -9256.394,E2 -9256.394} C_VEL
LIN {X 0,Y 432.627,Z 447.568,A -85,B 0,C 180,E1 -9258.046,E2 -9258.046} C_VEL
LIN {X 0,Y 431.99,Z 454.272,A -85,B 0,C 180,E1 -9259.691,E2 -9259.691} C_VEL
LIN {X 0,Y 431.629,Z 460.482,A -85,B 0,C 180,E1 -9261.573,E2 -9261.573} C_VEL
LIN {X 0,Y 431.373,Z 465.679,A -85,B 0,C 180,E1 -9263.629,E2 -9263.629} C_VEL
LIN {X 0,Y 431.243,Z 468.796,A -85,B 0,C 180,E1 -9265.326,E2 -9265.326} C_VEL
LIN {X 0,Y 431.23,Z 471.123,A -85,B 0,C 180,E1 -9267.198,E2 -9267.198} C_VEL
LIN {X 0,Y 431.146,Z 472.314,A -85,B 0,C 180,E1 -9269.066,E2 -9269.066} C_VEL
LIN {X 0,Y 431.147,Z 472.331,A -85,B 0,C 180,E1 -9270.934,E2 -9270.934} C_VEL
LIN {X 0,Y 431.23,Z 471.207,A -85,B 0,C 180,E1 -9272.803,E2 -9272.803} C_VEL
LIN {X 0,Y 431.238,Z 468.946,A -85,B 0,C 180,E1 -9274.674,E2 -9274.674} C_VEL
LIN {X 0,Y 431.336,Z 465.491,A -85,B 0,C 180,E1 -9276.549,E2 -9276.549} C_VEL
LIN {X 0,Y 431.602,Z 460.761,A -85,B 0,C 180,E1 -9278.427,E2 -9278.427} C_VEL
LIN {X 0,Y 431.965,Z 454.634,A -85,B 0,C 180,E1 -9280.31,E2 -9280.31} C_VEL
LIN {X 0,Y 432.565,Z 447.975,A -85,B 0,C 180,E1 -9281.956,E2 -9281.956} C_VEL
LIN {X 0,Y 433.137,Z 439.933,A -85,B 0,C 180,E1 -9283.608,E2 -9283.608} C_VEL
LIN {X 0,Y 434.028,Z 430.285,A -85,B 0,C 180,E1 -9285.256,E2 -9285.256} C_VEL
LIN {X 0,Y 434.942,Z 420.423,A -85,B 0,C 180,E1 -9286.667,E2 -9286.667} C_VEL
LIN {X 0,Y 436.032,Z 408.7,A -85,B 0,C 180,E1 -9288.075,E2 -9288.075} C_VEL
LIN {X 0,Y 437.256,Z 395.736,A -85,B 0,C 180,E1 -9289.36,E2 -9289.36} C_VEL
LIN {X 0,Y 438.327,Z 382.869,A -85,B 0,C 180,E1 -9290.41,E2 -9290.41} C_VEL
LIN {X 0,Y 439.422,Z 368.757,A -85,B 0,C 180,E1 -9291.337,E2 -9291.337} C_VEL
LIN {X 0,Y 440.345,Z 353.962,A -85,B 0,C 180,E1 -9292.096,E2 -9292.096} C_VEL
LIN {X 0,Y 441.015,Z 339.787,A -85,B 0,C 180,E1 -9292.641,E2 -9292.641} C_VEL
LIN {X 0,Y 441.525,Z 325.774,A -85,B 0,C 180,E1 -9293.015,E2 -9293.015} C_VEL
LIN {X 0,Y 443.671,Z 188.846,A -85,B 0,C 180,E1 -9295.297,E2 -9295.297} C_VEL
LIN {X 0,Y 438.82,Z 166.845,A -85,B 0,C 180,E1 -9295.989,E2 -9295.989} C_VEL
LIN {X 0,Y 436.881,Z 161.709,A -85,B 0,C 180,E1 -9296.248,E2 -9296.248} C_VEL
LIN {X 0,Y 433.726,Z 148.062,A -85,B 0,C 180,E1 -9298.954,E2 -9298.954} C_VEL
LIN {X 0,Y 432.391,Z 142.534,A -85,B 0,C 180,E1 -9300.122,E2 -9300.122} C_VEL
LIN {X 0,Y 432.331,Z 142.231,A -85,B 0,C 180,E1 -9300.506,E2 -9300.506} C_VEL
LIN {X 0,Y 432.333,Z 142.252,A -85,B 0,C 180,E1 -9303.998,E2 -9303.998} C_VEL
LIN {X 0,Y 432.312,Z 142.256,A -85,B 0,C 180,E1 -9307.195,E2 -9307.195} C_VEL
LIN {X 0,Y 432.289,Z 142.25,A -85,B 0,C 180,E1 -9310.172,E2 -9310.172} C_VEL
LIN {X 0,Y 432.303,Z 142.252,A -85,B 0,C 180,E1 -9313.063,E2 -9313.063} C_VEL
LIN {X 0,Y 432.332,Z 142.254,A -85,B 0,C 180,E1 -9315.665,E2 -9315.665} C_VEL
LIN {X 0,Y 432.308,Z 142.248,A -85,B 0,C 180,E1 -9318.402,E2 -9318.402} C_VEL
LIN {X 0,Y 432.328,Z 142.247,A -85,B 0,C 180,E1 -9321.849,E2 -9321.849} C_VEL
LIN {X 0,Y 432.328,Z 142.249,A -85,B 0,C 180,E1 -9325.322,E2 -9325.322} C_VEL
LIN {X 0,Y 432.316,Z 142.227,A -85,B 0,C 180,E1 -9328.653,E2 -9328.653} C_VEL
LIN {X 0,Y 432.329,Z 142.255,A -85,B 0,C 180,E1 -9331.873,E2 -9331.873} C_VEL
LIN {X 0,Y 432.355,Z 142.244,A -85,B 0,C 180,E1 -9335.546,E2 -9335.546} C_VEL
LIN {X 0,Y 432.351,Z 142.246,A -85,B 0,C 180,E1 -9339.046,E2 -9339.046} C_VEL
LIN {X 0,Y 432.351,Z 142.253,A -85,B 0,C 180,E1 -9342.01,E2 -9342.01} C_VEL
LIN {X 0,Y 432.352,Z 142.243,A -85,B 0,C 180,E1 -9344.925,E2 -9344.925} C_VEL
LIN {X 0,Y 432.461,Z 142.24,A -85,B 0,C 180,E1 -9347.803,E2 -9347.803} C_VEL
LIN {X 0,Y 432.465,Z 142.229,A -85,B 0,C 180,E1 -9351.59,E2 -9351.59} C_VEL
LIN {X 0,Y 432.587,Z 142.223,A -85,B 0,C 180,E1 -9354.406,E2 -9354.406} C_VEL
LIN {X 0,Y 432.6,Z 142.214,A -85,B 0,C 180,E1 -9358.138,E2 -9358.138} C_VEL
LIN {X 0,Y 432.728,Z 142.205,A -85,B 0,C 180,E1 -9360,E2 -9360} C_VEL
LIN {X 0,Y 432.585,Z 142.216,A -85,B 0,C 180,E1 -9362.794,E2 -9362.794} C_VEL
LIN {X 0,Y 432.587,Z 142.224,A -85,B 0,C 180,E1 -9365.594,E2 -9365.594} C_VEL
LIN {X 0,Y 432.466,Z 142.232,A -85,B 0,C 180,E1 -9368.41,E2 -9368.41} C_VEL
LIN {X 0,Y 432.461,Z 142.238,A -85,B 0,C 180,E1 -9372.196,E2 -9372.196} C_VEL
LIN {X 0,Y 432.432,Z 142.233,A -85,B 0,C 180,E1 -9376.039,E2 -9376.039} C_VEL
LIN {X 0,Y 432.388,Z 142.244,A -85,B 0,C 180,E1 -9379.485,E2 -9379.485} C_VEL
LIN {X 0,Y 432.318,Z 142.26,A -85,B 0,C 180,E1 -9382.964,E2 -9382.964} C_VEL
LIN {X 0,Y 432.351,Z 142.244,A -85,B 0,C 180,E1 -9386.033,E2 -9386.033} C_VEL
LIN {X 0,Y 432.344,Z 142.252,A -85,B 0,C 180,E1 -9389.187,E2 -9389.187} C_VEL
LIN {X 0,Y 432.322,Z 142.226,A -85,B 0,C 180,E1 -9392.443,E2 -9392.443} C_VEL
LIN {X 0,Y 432.338,Z 142.25,A -85,B 0,C 180,E1 -9395.818,E2 -9395.818} C_VEL
LIN {X 0,Y 432.347,Z 142.24,A -85,B 0,C 180,E1 -9399.343,E2 -9399.343} C_VEL
LIN {X 0,Y 432.334,Z 142.245,A -85,B 0,C 180,E1 -9401.797,E2 -9401.797} C_VEL
LIN {X 0,Y 432.334,Z 142.253,A -85,B 0,C 180,E1 -9404.347,E2 -9404.347} C_VEL
LIN {X 0,Y 432.321,Z 142.25,A -85,B 0,C 180,E1 -9407.016,E2 -9407.016} C_VEL
LIN {X 0,Y 432.334,Z 142.249,A -85,B 0,C 180,E1 -9409.821,E2 -9409.821} C_VEL
LIN {X 0,Y 432.311,Z 142.258,A -85,B 0,C 180,E1 -9413.022,E2 -9413.022} C_VEL
LIN {X 0,Y 432.36,Z 142.25,A -85,B 0,C 180,E1 -9415.996,E2 -9415.996} C_VEL
LIN {X 0,Y 432.388,Z 142.401,A -85,B 0,C 180,E1 -9418.789,E2 -9418.789} C_VEL
LIN {X 0,Y 435.909,Z 156.489,A -85,B 0,C 180,E1 -9421.6,E2 -9421.6} C_VEL
LIN {X 0,Y 437.782,Z 165.45,A -85,B 0,C 180,E1 -9423.288,E2 -9423.288} C_VEL
LIN {X 0,Y 437.646,Z 169.286,A -85,B 0,C 180,E1 -9423.877,E2 -9423.877} C_VEL
LIN {X 0,Y 443.421,Z 196.93,A -85,B 0,C 180,E1 -9424.744,E2 -9424.744} C_VEL
LIN {X 0,Y 442.437,Z 272.865,A -85,B 0,C 180,E1 -9426.012,E2 -9426.012} C_VEL
LIN {X 0,Y 441.392,Z 335.501,A -85,B 0,C 180,E1 -9427.07,E2 -9427.07} C_VEL
LIN {X 0,Y 440.754,Z 351.042,A -85,B 0,C 180,E1 -9427.518,E2 -9427.518} C_VEL
LIN {X 0,Y 439.997,Z 365.055,A -85,B 0,C 180,E1 -9428.095,E2 -9428.095} C_VEL
LIN {X 0,Y 439.014,Z 379.656,A -85,B 0,C 180,E1 -9428.888,E2 -9428.888} C_VEL
LIN {X 0,Y 437.896,Z 393.13,A -85,B 0,C 180,E1 -9429.814,E2 -9429.814} C_VEL
LIN {X 0,Y 436.723,Z 406.846,A -85,B 0,C 180,E1 -9430.981,E2 -9430.981} C_VEL
LIN {X 0,Y 435.559,Z 419.719,A -85,B 0,C 180,E1 -9432.322,E2 -9432.322} C_VEL
LIN {X 0,Y 434.422,Z 431.427,A -85,B 0,C 180,E1 -9433.795,E2 -9433.795} C_VEL
LIN {X 0,Y 433.491,Z 442.245,A -85,B 0,C 180,E1 -9435.446,E2 -9435.446} C_VEL
LIN {X 0,Y 432.677,Z 451.056,A -85,B 0,C 180,E1 -9437.054,E2 -9437.054} C_VEL
LIN {X 0,Y 432.196,Z 458.723,A -85,B 0,C 180,E1 -9438.747,E2 -9438.747} C_VEL
LIN {X 0,Y 431.664,Z 465.69,A -85,B 0,C 180,E1 -9440.63,E2 -9440.63} C_VEL
LIN {X 0,Y 431.407,Z 471.168,A -85,B 0,C 180,E1 -9442.511,E2 -9442.511} C_VEL
LIN {X 0,Y 431.253,Z 475.308,A -85,B 0,C 180,E1 -9444.389,E2 -9444.389} C_VEL
LIN {X 0,Y 431.137,Z 478.21,A -85,B 0,C 180,E1 -9446.261,E2 -9446.261} C_VEL
LIN {X 0,Y 431.193,Z 479.941,A -85,B 0,C 180,E1 -9448.132,E2 -9448.132} C_VEL
LIN {X 0,Y 431.141,Z 480.534,A -85,B 0,C 180,E1 -9450,E2 -9450} C_VEL
LIN {X 0,Y 431.193,Z 479.937,A -85,B 0,C 180,E1 -9451.868,E2 -9451.868} C_VEL
LIN {X 0,Y 431.138,Z 478.201,A -85,B 0,C 180,E1 -9453.739,E2 -9453.739} C_VEL
LIN {X 0,Y 431.266,Z 475.3,A -85,B 0,C 180,E1 -9455.611,E2 -9455.611} C_VEL
LIN {X 0,Y 431.408,Z 471.162,A -85,B 0,C 180,E1 -9457.488,E2 -9457.488} C_VEL
LIN {X 0,Y 431.664,Z 465.678,A -85,B 0,C 180,E1 -9459.37,E2 -9459.37} C_VEL
LIN {X 0,Y 432.196,Z 458.7,A -85,B 0,C 180,E1 -9461.253,E2 -9461.253} C_VEL
LIN {X 0,Y 432.753,Z 450.011,A -85,B 0,C 180,E1 -9463.142,E2 -9463.142} C_VEL
LIN {X 0,Y 433.616,Z 440.781,A -85,B 0,C 180,E1 -9464.79,E2 -9464.79} C_VEL
LIN {X 0,Y 434.458,Z 431.394,A -85,B 0,C 180,E1 -9466.203,E2 -9466.203} C_VEL
LIN {X 0,Y 435.511,Z 419.866,A -85,B 0,C 180,E1 -9467.658,E2 -9467.658} C_VEL
LIN {X 0,Y 436.739,Z 406.802,A -85,B 0,C 180,E1 -9469.018,E2 -9469.018} C_VEL
LIN {X 0,Y 437.889,Z 393.059,A -85,B 0,C 180,E1 -9470.186,E2 -9470.186} C_VEL
LIN {X 0,Y 439.031,Z 379.561,A -85,B 0,C 180,E1 -9471.111,E2 -9471.111} C_VEL
LIN {X 0,Y 439.989,Z 365.046,A -85,B 0,C 180,E1 -9471.901,E2 -9471.901} C_VEL
LIN {X 0,Y 440.758,Z 350.451,A -85,B 0,C 180,E1 -9472.5,E2 -9472.5} C_VEL
LIN {X 0,Y 441.361,Z 335.29,A -85,B 0,C 180,E1 -9472.931,E2 -9472.931} C_VEL
LIN {X 0,Y 443.534,Z 198.287,A -85,B 0,C 180,E1 -9475.219,E2 -9475.219} C_VEL
LIN {X 0,Y 438.517,Z 173.418,A -85,B 0,C 180,E1 -9475.97,E2 -9475.97} C_VEL
LIN {X 0,Y 437.598,Z 168.86,A -85,B 0,C 180,E1 -9476.153,E2 -9476.153} C_VEL
LIN {X 0,Y 437.744,Z 165.408,A -85,B 0,C 180,E1 -9476.714,E2 -9476.714} C_VEL
LIN {X 0,Y 435.158,Z 153.461,A -85,B 0,C 180,E1 -9478.981,E2 -9478.981} C_VEL
LIN {X 0,Y 432.356,Z 142.328,A -85,B 0,C 180,E1 -9481.239,E2 -9481.239} C_VEL
LIN {X 0,Y 432.34,Z 142.257,A -85,B 0,C 180,E1 -9484.677,E2 -9484.677} C_VEL
LIN {X 0,Y 432.343,Z 142.253,A -85,B 0,C 180,E1 -9488.149,E2 -9488.149} C_VEL
LIN {X 0,Y 432.333,Z 142.259,A -85,B 0,C 180,E1 -9491.602,E2 -9491.602} C_VEL
LIN {X 0,Y 432.334,Z 142.243,A -85,B 0,C 180,E1 -9494.347,E2 -9494.347} C_VEL
LIN {X 0,Y 432.32,Z 142.257,A -85,B 0,C 180,E1 -9497.016,E2 -9497.016} C_VEL
LIN {X 0,Y 432.333,Z 142.236,A -85,B 0,C 180,E1 -9499.821,E2 -9499.821} C_VEL
LIN {X 0,Y 432.307,Z 142.259,A -85,B 0,C 180,E1 -9503.022,E2 -9503.022} C_VEL
LIN {X 0,Y 432.333,Z 142.228,A -85,B 0,C 180,E1 -9506.002,E2 -9506.002} C_VEL
LIN {X 0,Y 432.348,Z 142.245,A -85,B 0,C 180,E1 -9509.49,E2 -9509.49} C_VEL
LIN {X 0,Y 432.392,Z 142.247,A -85,B 0,C 180,E1 -9512.928,E2 -9512.928} C_VEL
LIN {X 0,Y 432.371,Z 142.249,A -85,B 0,C 180,E1 -9516.023,E2 -9516.023} C_VEL
LIN {X 0,Y 432.351,Z 142.246,A -85,B 0,C 180,E1 -9519.046,E2 -9519.046} C_VEL
LIN {X 0,Y 432.361,Z 142.25,A -85,B 0,C 180,E1 -9522.011,E2 -9522.011} C_VEL
LIN {X 0,Y 432.395,Z 142.24,A -85,B 0,C 180,E1 -9524.927,E2 -9524.927} C_VEL
LIN {X 0,Y 432.461,Z 142.238,A -85,B 0,C 180,E1 -9527.804,E2 -9527.804} C_VEL
LIN {X 0,Y 432.465,Z 142.233,A -85,B 0,C 180,E1 -9531.59,E2 -9531.59} C_VEL
LIN {X 0,Y 432.587,Z 142.225,A -85,B 0,C 180,E1 -9534.406,E2 -9534.406} C_VEL
LIN {X 0,Y 432.604,Z 142.216,A -85,B 0,C 180,E1 -9538.138,E2 -9538.138} C_VEL
LIN {X 0,Y 432.73,Z 142.205,A -85,B 0,C 180,E1 -9540,E2 -9540} C_VEL
LIN {X 0,Y 432.58,Z 142.215,A -85,B 0,C 180,E1 -9542.794,E2 -9542.794} C_VEL
LIN {X 0,Y 432.587,Z 142.222,A -85,B 0,C 180,E1 -9545.594,E2 -9545.594} C_VEL
LIN {X 0,Y 432.465,Z 142.229,A -85,B 0,C 180,E1 -9548.41,E2 -9548.41} C_VEL
LIN {X 0,Y 432.461,Z 142.241,A -85,B 0,C 180,E1 -9552.197,E2 -9552.197} C_VEL
LIN {X 0,Y 432.419,Z 142.242,A -85,B 0,C 180,E1 -9556.039,E2 -9556.039} C_VEL
LIN {X 0,Y 432.388,Z 142.243,A -85,B 0,C 180,E1 -9559.485,E2 -9559.485} C_VEL
LIN {X 0,Y 432.314,Z 142.256,A -85,B 0,C 180,E1 -9562.965,E2 -9562.965} C_VEL
LIN {X 0,Y 432.318,Z 142.254,A -85,B 0,C 180,E1 -9566.036,E2 -9566.036} C_VEL
LIN {X 0,Y 432.327,Z 142.255,A -85,B 0,C 180,E1 -9569.189,E2 -9569.189} C_VEL
LIN {X 0,Y 432.321,Z 142.222,A -85,B 0,C 180,E1 -9572.443,E2 -9572.443} C_VEL
LIN {X 0,Y 432.337,Z 142.258,A -85,B 0,C 180,E1 -9575.818,E2 -9575.818} C_VEL
LIN {X 0,Y 432.302,Z 142.236,A -85,B 0,C 180,E1 -9579.348,E2 -9579.348} C_VEL
LIN {X 0,Y 432.304,Z 142.25,A -85,B 0,C 180,E1 -9581.801,E2 -9581.801} C_VEL
LIN {X 0,Y 432.334,Z 142.254,A -85,B 0,C 180,E1 -9584.347,E2 -9584.347} C_VEL
LIN {X 0,Y 432.303,Z 142.252,A -85,B 0,C 180,E1 -9587.018,E2 -9587.018} C_VEL
LIN {X 0,Y 432.29,Z 142.251,A -85,B 0,C 180,E1 -9589.828,E2 -9589.828} C_VEL
LIN {X 0,Y 432.304,Z 142.255,A -85,B 0,C 180,E1 -9593.022,E2 -9593.022} C_VEL
LIN {X 0,Y 432.333,Z 142.253,A -85,B 0,C 180,E1 -9596.002,E2 -9596.002} C_VEL
LIN {X 0,Y 432.331,Z 142.231,A -85,B 0,C 180,E1 -9599.494,E2 -9599.494} C_VEL
LIN {X 0,Y 432.342,Z 142.284,A -85,B 0,C 180,E1 -9599.875,E2 -9599.875} C_VEL
LIN {X 0,Y 432.763,Z 143.997,A -85,B 0,C 180,E1 -9600.309,E2 -9600.309} C_VEL
LIN {X 0,Y 435.671,Z 156.222,A -85,B 0,C 180,E1 -9602.791,E2 -9602.791} C_VEL
LIN {X 0,Y 436.983,Z 162.115,A -85,B 0,C 180,E1 -9603.89,E2 -9603.89} C_VEL
LIN {X 0,Y 439.076,Z 167.685,A -85,B 0,C 180,E1 -9604.14,E2 -9604.14} C_VEL
LIN {X 0,Y 443.624,Z 189.073,A -85,B 0,C 180,E1 -9604.801,E2 -9604.801} C_VEL
LIN {X 0,Y 441.537,Z 324.128,A -85,B 0,C 180,E1 -9607.047,E2 -9607.047} C_VEL
LIN {X 0,Y 441.004,Z 339.713,A -85,B 0,C 180,E1 -9607.451,E2 -9607.451} C_VEL
LIN {X 0,Y 440.306,Z 354.225,A -85,B 0,C 180,E1 -9608.009,E2 -9608.009} C_VEL
LIN {X 0,Y 439.367,Z 369.194,A -85,B 0,C 180,E1 -9608.783,E2 -9608.783} C_VEL
LIN {X 0,Y 439.296,Z 370.475,A -85,B 0,C 180,E1 -9608.859,E2 -9608.859} C_VEL
LIN {X 0,Y 438.321,Z 375.826,A -85,B 0,C 180,E1 -9609.161,E2 -9609.161} C_VEL
LIN {X 0,Y 434.89,Z 384.416,A -85,B 0,C 180,E1 -9609.635,E2 -9609.635} C_VEL
LIN {X 0,Y 431.414,Z 392.786,A -85,B 0,C 180,E1 -9610.176,E2 -9610.176} C_VEL
LIN {X 0,Y 430.348,Z 397.651,A -85,B 0,C 180,E1 -9610.59,E2 -9610.59} C_VEL
LIN {X 0,Y 429.145,Z 410.071,A -85,B 0,C 180,E1 -9611.871,E2 -9611.871} C_VEL
LIN {X 0,Y 428.005,Z 421.573,A -85,B 0,C 180,E1 -9613.3,E2 -9613.3} C_VEL
LIN {X 0,Y 427.071,Z 431.253,A -85,B 0,C 180,E1 -9614.734,E2 -9614.734} C_VEL
LIN {X 0,Y 426.125,Z 440.743,A -85,B 0,C 180,E1 -9616.407,E2 -9616.407} C_VEL
LIN {X 0,Y 425.534,Z 448.643,A -85,B 0,C 180,E1 -9618.086,E2 -9618.086} C_VEL
LIN {X 0,Y 424.865,Z 456.023,A -85,B 0,C 180,E1 -9619.998,E2 -9619.998} C_VEL
LIN {X 0,Y 424.488,Z 461.879,A -85,B 0,C 180,E1 -9621.91,E2 -9621.91} C_VEL
LIN {X 0,Y 424.295,Z 466,A -85,B 0,C 180,E1 -9623.636,E2 -9623.636} C_VEL
LIN {X 0,Y 424.172,Z 468.863,A -85,B 0,C 180,E1 -9625.248,E2 -9625.248} C_VEL
LIN {X 0,Y 424.126,Z 471.19,A -85,B 0,C 180,E1 -9627.151,E2 -9627.151} C_VEL
LIN {X 0,Y 424.067,Z 472.38,A -85,B 0,C 180,E1 -9629.05,E2 -9629.05} C_VEL
LIN {X 0,Y 424.068,Z 472.397,A -85,B 0,C 180,E1 -9630.95,E2 -9630.95} C_VEL
LIN {X 0,Y 424.126,Z 471.273,A -85,B 0,C 180,E1 -9632.849,E2 -9632.849} C_VEL
LIN {X 0,Y 424.167,Z 469.011,A -85,B 0,C 180,E1 -9634.752,E2 -9634.752} C_VEL
LIN {X 0,Y 424.251,Z 465.556,A -85,B 0,C 180,E1 -9636.659,E2 -9636.659} C_VEL
LIN {X 0,Y 424.563,Z 460.826,A -85,B 0,C 180,E1 -9638.568,E2 -9638.568} C_VEL
LIN {X 0,Y 424.935,Z 454.699,A -85,B 0,C 180,E1 -9640.482,E2 -9640.482} C_VEL
LIN {X 0,Y 425.557,Z 448.04,A -85,B 0,C 180,E1 -9642.155,E2 -9642.155} C_VEL
LIN {X 0,Y 426.176,Z 439.998,A -85,B 0,C 180,E1 -9643.835,E2 -9643.835} C_VEL
LIN {X 0,Y 427.137,Z 430.349,A -85,B 0,C 180,E1 -9645.508,E2 -9645.508} C_VEL
LIN {X 0,Y 428.105,Z 420.486,A -85,B 0,C 180,E1 -9646.942,E2 -9646.942} C_VEL
LIN {X 0,Y 429.262,Z 408.762,A -85,B 0,C 180,E1 -9648.37,E2 -9648.37} C_VEL
LIN {X 0,Y 430.551,Z 395.798,A -85,B 0,C 180,E1 -9649.674,E2 -9649.674} C_VEL
LIN {X 0,Y 431.674,Z 382.929,A -85,B 0,C 180,E1 -9650.739,E2 -9650.739} C_VEL
LIN {X 0,Y 432.814,Z 368.816,A -85,B 0,C 180,E1 -9651.679,E2 -9651.679} C_VEL
LIN {X 0,Y 433.76,Z 354.293,A -85,B 0,C 180,E1 -9652.437,E2 -9652.437} C_VEL
LIN {X 0,Y 434.47,Z 339.84,A -85,B 0,C 180,E1 -9653.001,E2 -9653.001} C_VEL
LIN {X 0,Y 435.004,Z 325.818,A -85,B 0,C 180,E1 -9653.381,E2 -9653.381} C_VEL
LIN {X 0,Y 437.304,Z 190.571,A -85,B 0,C 180,E1 -9655.661,E2 -9655.661} C_VEL
LIN {X 0,Y 432.766,Z 169.495,A -85,B 0,C 180,E1 -9656.333,E2 -9656.333} C_VEL
LIN {X 0,Y 429.708,Z 161.946,A -85,B 0,C 180,E1 -9656.704,E2 -9656.704} C_VEL
LIN {X 0,Y 427.067,Z 150.463,A -85,B 0,C 180,E1 -9659.004,E2 -9659.004} C_VEL
LIN {X 0,Y 425.333,Z 143.344,A -85,B 0,C 180,E1 -9660.537,E2 -9660.537} C_VEL
LIN {X 0,Y 425.282,Z 143.11,A -85,B 0,C 180,E1 -9660.817,E2 -9660.817} C_VEL
LIN {X 0,Y 425.291,Z 143.131,A -85,B 0,C 180,E1 -9664.284,E2 -9664.284} C_VEL
LIN {X 0,Y 425.271,Z 143.138,A -85,B 0,C 180,E1 -9667.695,E2 -9667.695} C_VEL
LIN {X 0,Y 425.243,Z 143.129,A -85,B 0,C 180,E1 -9670.514,E2 -9670.514} C_VEL
LIN {X 0,Y 425.246,Z 143.128,A -85,B 0,C 180,E1 -9673.349,E2 -9673.349} C_VEL
LIN {X 0,Y 425.257,Z 143.135,A -85,B 0,C 180,E1 -9676.043,E2 -9676.043} C_VEL
LIN {X 0,Y 425.248,Z 143.122,A -85,B 0,C 180,E1 -9678.618,E2 -9678.618} C_VEL
LIN {X 0,Y 425.28,Z 143.115,A -85,B 0,C 180,E1 -9681.099,E2 -9681.099} C_VEL
LIN {X 0,Y 425.296,Z 143.131,A -85,B 0,C 180,E1 -9684.664,E2 -9684.664} C_VEL
LIN {X 0,Y 425.261,Z 143.1,A -85,B 0,C 180,E1 -9688.073,E2 -9688.073} C_VEL
LIN {X 0,Y 425.306,Z 143.128,A -85,B 0,C 180,E1 -9691.366,E2 -9691.366} C_VEL
LIN {X 0,Y 425.261,Z 143.128,A -85,B 0,C 180,E1 -9694.552,E2 -9694.552} C_VEL
LIN {X 0,Y 425.294,Z 143.133,A -85,B 0,C 180,E1 -9697.73,E2 -9697.73} C_VEL
LIN {X 0,Y 425.362,Z 143.118,A -85,B 0,C 180,E1 -9700.704,E2 -9700.704} C_VEL
LIN {X 0,Y 425.325,Z 143.13,A -85,B 0,C 180,E1 -9703.686,E2 -9703.686} C_VEL
LIN {X 0,Y 425.396,Z 143.114,A -85,B 0,C 180,E1 -9707.096,E2 -9707.096} C_VEL
LIN {X 0,Y 425.399,Z 143.11,A -85,B 0,C 180,E1 -9710.49,E2 -9710.49} C_VEL
LIN {X 0,Y 425.5,Z 143.103,A -85,B 0,C 180,E1 -9713.361,E2 -9713.361} C_VEL
LIN {X 0,Y 425.357,Z 143.125,A -85,B 0,C 180,E1 -9715.261,E2 -9715.261} C_VEL
LIN {X 0,Y 425.569,Z 143.088,A -85,B 0,C 180,E1 -9718.107,E2 -9718.107} C_VEL
LIN {X 0,Y 425.697,Z 143.081,A -85,B 0,C 180,E1 -9720,E2 -9720} C_VEL
LIN {X 0,Y 425.538,Z 143.094,A -85,B 0,C 180,E1 -9722.84,E2 -9722.84} C_VEL
LIN {X 0,Y 425.543,Z 143.102,A -85,B 0,C 180,E1 -9725.687,E2 -9725.687} C_VEL
LIN {X 0,Y 425.41,Z 143.112,A -85,B 0,C 180,E1 -9728.551,E2 -9728.551} C_VEL
LIN {X 0,Y 425.414,Z 143.116,A -85,B 0,C 180,E1 -9732.402,E2 -9732.402} C_VEL
LIN {X 0,Y 425.389,Z 143.111,A -85,B 0,C 180,E1 -9736.312,E2 -9736.312} C_VEL
LIN {X 0,Y 425.33,Z 143.122,A -85,B 0,C 180,E1 -9739.635,E2 -9739.635} C_VEL
LIN {X 0,Y 425.289,Z 143.128,A -85,B 0,C 180,E1 -9742.339,E2 -9742.339} C_VEL
LIN {X 0,Y 425.321,Z 143.129,A -85,B 0,C 180,E1 -9744.657,E2 -9744.657} C_VEL
LIN {X 0,Y 425.347,Z 143.124,A -85,B 0,C 180,E1 -9747.558,E2 -9747.558} C_VEL
LIN {X 0,Y 425.289,Z 143.118,A -85,B 0,C 180,E1 -9750.816,E2 -9750.816} C_VEL
LIN {X 0,Y 425.292,Z 143.109,A -85,B 0,C 180,E1 -9754.284,E2 -9754.284} C_VEL
LIN {X 0,Y 425.28,Z 143.133,A -85,B 0,C 180,E1 -9757.694,E2 -9757.694} C_VEL
LIN {X 0,Y 425.28,Z 143.113,A -85,B 0,C 180,E1 -9760.52,E2 -9760.52} C_VEL
LIN {X 0,Y 425.258,Z 143.137,A -85,B 0,C 180,E1 -9763.351,E2 -9763.351} C_VEL
LIN {X 0,Y 425.258,Z 143.124,A -85,B 0,C 180,E1 -9766.649,E2 -9766.649} C_VEL
LIN {X 0,Y 425.286,Z 143.125,A -85,B 0,C 180,E1 -9769.872,E2 -9769.872} C_VEL
LIN {X 0,Y 425.282,Z 143.136,A -85,B 0,C 180,E1 -9772.488,E2 -9772.488} C_VEL
LIN {X 0,Y 425.308,Z 143.131,A -85,B 0,C 180,E1 -9775.817,E2 -9775.817} C_VEL
LIN {X 0,Y 425.321,Z 143.282,A -85,B 0,C 180,E1 -9778.391,E2 -9778.391} C_VEL
LIN {X 0,Y 429.003,Z 157.915,A -85,B 0,C 180,E1 -9781.368,E2 -9781.368} C_VEL
LIN {X 0,Y 430.894,Z 166.724,A -85,B 0,C 180,E1 -9783.062,E2 -9783.062} C_VEL
LIN {X 0,Y 430.955,Z 169.097,A -85,B 0,C 180,E1 -9783.434,E2 -9783.434} C_VEL
LIN {X 0,Y 436.138,Z 193.69,A -85,B 0,C 180,E1 -9784.234,E2 -9784.234} C_VEL
LIN {X 0,Y 437.122,Z 199.143,A -85,B 0,C 180,E1 -9784.394,E2 -9784.394} C_VEL
LIN {X 0,Y 434.911,Z 334.141,A -85,B 0,C 180,E1 -9786.677,E2 -9786.677} C_VEL
LIN {X 0,Y 434.253,Z 349.668,A -85,B 0,C 180,E1 -9787.112,E2 -9787.112} C_VEL
LIN {X 0,Y 433.492,Z 363.718,A -85,B 0,C 180,E1 -9787.687,E2 -9787.687} C_VEL
LIN {X 0,Y 432.531,Z 377.607,A -85,B 0,C 180,E1 -9788.431,E2 -9788.431} C_VEL
LIN {X 0,Y 431.328,Z 391.485,A -85,B 0,C 180,E1 -9789.369,E2 -9789.369} C_VEL
LIN {X 0,Y 430.208,Z 404.199,A -85,B 0,C 180,E1 -9790.434,E2 -9790.434} C_VEL
LIN {X 0,Y 429,Z 417.053,A -85,B 0,C 180,E1 -9791.741,E2 -9791.741} C_VEL
LIN {X 0,Y 427.942,Z 427.813,A -85,B 0,C 180,E1 -9793.052,E2 -9793.052} C_VEL
LIN {X 0,Y 426.945,Z 437.767,A -85,B 0,C 180,E1 -9794.485,E2 -9794.485} C_VEL
LIN {X 0,Y 426.025,Z 447.503,A -85,B 0,C 180,E1 -9796.16,E2 -9796.16} C_VEL
LIN {X 0,Y 425.365,Z 455.627,A -85,B 0,C 180,E1 -9797.839,E2 -9797.839} C_VEL
LIN {X 0,Y 424.796,Z 462.339,A -85,B 0,C 180,E1 -9799.514,E2 -9799.514} C_VEL
LIN {X 0,Y 424.466,Z 468.539,A -85,B 0,C 180,E1 -9801.43,E2 -9801.43} C_VEL
LIN {X 0,Y 424.243,Z 473.332,A -85,B 0,C 180,E1 -9803.341,E2 -9803.341} C_VEL
LIN {X 0,Y 424.144,Z 476.844,A -85,B 0,C 180,E1 -9805.248,E2 -9805.248} C_VEL
LIN {X 0,Y 424.073,Z 479.153,A -85,B 0,C 180,E1 -9807.15,E2 -9807.15} C_VEL
LIN {X 0,Y 424.066,Z 480.315,A -85,B 0,C 180,E1 -9809.05,E2 -9809.05} C_VEL
LIN {X 0,Y 424.066,Z 480.313,A -85,B 0,C 180,E1 -9810.95,E2 -9810.95} C_VEL
LIN {X 0,Y 424.073,Z 479.145,A -85,B 0,C 180,E1 -9812.85,E2 -9812.85} C_VEL
LIN {X 0,Y 424.147,Z 476.833,A -85,B 0,C 180,E1 -9814.752,E2 -9814.752} C_VEL
LIN {X 0,Y 424.293,Z 473.324,A -85,B 0,C 180,E1 -9816.658,E2 -9816.658} C_VEL
LIN {X 0,Y 424.466,Z 468.53,A -85,B 0,C 180,E1 -9818.57,E2 -9818.57} C_VEL
LIN {X 0,Y 424.796,Z 462.318,A -85,B 0,C 180,E1 -9820.486,E2 -9820.486} C_VEL
LIN {X 0,Y 425.355,Z 455.6,A -85,B 0,C 180,E1 -9822.161,E2 -9822.161} C_VEL
LIN {X 0,Y 426.124,Z 446.219,A -85,B 0,C 180,E1 -9824.08,E2 -9824.08} C_VEL
LIN {X 0,Y 427.096,Z 436.219,A -85,B 0,C 180,E1 -9825.754,E2 -9825.754} C_VEL
LIN {X 0,Y 428.156,Z 425.99,A -85,B 0,C 180,E1 -9827.185,E2 -9827.185} C_VEL
LIN {X 0,Y 429.319,Z 413.798,A -85,B 0,C 180,E1 -9828.616,E2 -9828.616} C_VEL
LIN {X 0,Y 430.464,Z 401.559,A -85,B 0,C 180,E1 -9829.802,E2 -9829.802} C_VEL
LIN {X 0,Y 431.603,Z 388.236,A -85,B 0,C 180,E1 -9830.867,E2 -9830.867} C_VEL
LIN {X 0,Y 432.861,Z 373.529,A -85,B 0,C 180,E1 -9831.802,E2 -9831.802} C_VEL
LIN {X 0,Y 433.747,Z 358.475,A -85,B 0,C 180,E1 -9832.546,E2 -9832.546} C_VEL
LIN {X 0,Y 434.535,Z 343.083,A -85,B 0,C 180,E1 -9833.092,E2 -9833.092} C_VEL
LIN {X 0,Y 435.009,Z 327.808,A -85,B 0,C 180,E1 -9833.443,E2 -9833.443} C_VEL
LIN {X 0,Y 437.11,Z 199.198,A -85,B 0,C 180,E1 -9835.599,E2 -9835.599} C_VEL
LIN {X 0,Y 431.971,Z 173.929,A -85,B 0,C 180,E1 -9836.383,E2 -9836.383} C_VEL
LIN {X 0,Y 430.925,Z 168.881,A -85,B 0,C 180,E1 -9836.578,E2 -9836.578} C_VEL
LIN {X 0,Y 430.639,Z 165.334,A -85,B 0,C 180,E1 -9837.191,E2 -9837.191} C_VEL
LIN {X 0,Y 427.87,Z 153.388,A -85,B 0,C 180,E1 -9839.523,E2 -9839.523} C_VEL
LIN {X 0,Y 425.294,Z 143.193,A -85,B 0,C 180,E1 -9841.646,E2 -9841.646} C_VEL
LIN {X 0,Y 425.312,Z 143.134,A -85,B 0,C 180,E1 -9844.288,E2 -9844.288} C_VEL
LIN {X 0,Y 425.283,Z 143.137,A -85,B 0,C 180,E1 -9847.694,E2 -9847.694} C_VEL
LIN {X 0,Y 425.28,Z 143.132,A -85,B 0,C 180,E1 -9850.52,E2 -9850.52} C_VEL
LIN {X 0,Y 425.257,Z 143.124,A -85,B 0,C 180,E1 -9853.351,E2 -9853.351} C_VEL
LIN {X 0,Y 425.258,Z 143.137,A -85,B 0,C 180,E1 -9856.649,E2 -9856.649} C_VEL
LIN {X 0,Y 425.286,Z 143.113,A -85,B 0,C 180,E1 -9859.873,E2 -9859.873} C_VEL
LIN {X 0,Y 425.278,Z 143.133,A -85,B 0,C 180,E1 -9862.489,E2 -9862.489} C_VEL
LIN {X 0,Y 425.286,Z 143.107,A -85,B 0,C 180,E1 -9865.816,E2 -9865.816} C_VEL
LIN {X 0,Y 425.291,Z 143.119,A -85,B 0,C 180,E1 -9869.239,E2 -9869.239} C_VEL
LIN {X 0,Y 425.349,Z 143.123,A -85,B 0,C 180,E1 -9872.442,E2 -9872.442} C_VEL
LIN {X 0,Y 425.351,Z 143.126,A -85,B 0,C 180,E1 -9875.602,E2 -9875.602} C_VEL
LIN {X 0,Y 425.294,Z 143.125,A -85,B 0,C 180,E1 -9878.682,E2 -9878.682} C_VEL
LIN {X 0,Y 425.322,Z 143.128,A -85,B 0,C 180,E1 -9881.702,E2 -9881.702} C_VEL
LIN {X 0,Y 425.348,Z 143.115,A -85,B 0,C 180,E1 -9884.671,E2 -9884.671} C_VEL
LIN {X 0,Y 425.414,Z 143.116,A -85,B 0,C 180,E1 -9887.598,E2 -9887.598} C_VEL
LIN {X 0,Y 425.409,Z 143.112,A -85,B 0,C 180,E1 -9891.449,E2 -9891.449} C_VEL
LIN {X 0,Y 425.543,Z 143.102,A -85,B 0,C 180,E1 -9894.313,E2 -9894.313} C_VEL
LIN {X 0,Y 425.574,Z 143.091,A -85,B 0,C 180,E1 -9898.107,E2 -9898.107} C_VEL
LIN {X 0,Y 425.699,Z 143.081,A -85,B 0,C 180,E1 -9900,E2 -9900} C_VEL
LIN {X 0,Y 425.533,Z 143.092,A -85,B 0,C 180,E1 -9902.84,E2 -9902.84} C_VEL
LIN {X 0,Y 425.499,Z 143.103,A -85,B 0,C 180,E1 -9906.517,E2 -9906.517} C_VEL
LIN {X 0,Y 425.4,Z 143.11,A -85,B 0,C 180,E1 -9909.51,E2 -9909.51} C_VEL
LIN {X 0,Y 425.395,Z 143.115,A -85,B 0,C 180,E1 -9912.904,E2 -9912.904} C_VEL
LIN {X 0,Y 425.347,Z 143.125,A -85,B 0,C 180,E1 -9916.597,E2 -9916.597} C_VEL
LIN {X 0,Y 425.33,Z 143.12,A -85,B 0,C 180,E1 -9919.635,E2 -9919.635} C_VEL
LIN {X 0,Y 425.289,Z 143.133,A -85,B 0,C 180,E1 -9922.339,E2 -9922.339} C_VEL
LIN {X 0,Y 425.26,Z 143.128,A -85,B 0,C 180,E1 -9925.448,E2 -9925.448} C_VEL
LIN {X 0,Y 425.308,Z 143.128,A -85,B 0,C 180,E1 -9928.86,E2 -9928.86} C_VEL
LIN {X 0,Y 425.261,Z 143.1,A -85,B 0,C 180,E1 -9931.927,E2 -9931.927} C_VEL
LIN {X 0,Y 425.295,Z 143.129,A -85,B 0,C 180,E1 -9935.336,E2 -9935.336} C_VEL
LIN {X 0,Y 425.281,Z 143.117,A -85,B 0,C 180,E1 -9938.901,E2 -9938.901} C_VEL
LIN {X 0,Y 425.257,Z 143.134,A -85,B 0,C 180,E1 -9942.655,E2 -9942.655} C_VEL
LIN {X 0,Y 425.285,Z 143.122,A -85,B 0,C 180,E1 -9945.283,E2 -9945.283} C_VEL
LIN {X 0,Y 425.248,Z 143.14,A -85,B 0,C 180,E1 -9948.618,E2 -9948.618} C_VEL
LIN {X 0,Y 425.281,Z 143.129,A -85,B 0,C 180,E1 -9951.099,E2 -9951.099} C_VEL
LIN {X 0,Y 425.295,Z 143.132,A -85,B 0,C 180,E1 -9954.664,E2 -9954.664} C_VEL
LIN {X 0,Y 425.255,Z 143.136,A -85,B 0,C 180,E1 -9958.072,E2 -9958.072} C_VEL
LIN {X 0,Y 425.305,Z 143.178,A -85,B 0,C 180,E1 -9959.489,E2 -9959.489} C_VEL
LIN {X 0,Y 425.847,Z 145.483,A -85,B 0,C 180,E1 -9960.051,E2 -9960.051} C_VEL
LIN {X 0,Y 428.918,Z 158.25,A -85,B 0,C 180,E1 -9962.691,E2 -9962.691} C_VEL
LIN {X 0,Y 429.795,Z 162.153,A -85,B 0,C 180,E1 -9963.417,E2 -9963.417} C_VEL
LIN {X 0,Y 433.018,Z 170.392,A -85,B 0,C 180,E1 -9963.798,E2 -9963.798} C_VEL
LIN {X 0,Y 437.102,Z 189.276,A -85,B 0,C 180,E1 -9964.4,E2 -9964.4} C_VEL
LIN {X 0,Y 435.638,Z 289.286,A -85,B 0,C 180,E1 -9966.088,E2 -9966.088} C_VEL
LIN {X 0,Y 434.932,Z 328.398,A -85,B 0,C 180,E1 -9966.773,E2 -9966.773} C_VEL
LIN {X 0,Y 434.263,Z 343.932,A -85,B 0,C 180,E1 -9967.232,E2 -9967.232} C_VEL
LIN {X 0,Y 433.566,Z 357.856,A -85,B 0,C 180,E1 -9967.822,E2 -9967.822} C_VEL
LIN {X 0,Y 432.638,Z 371.251,A -85,B 0,C 180,E1 -9968.562,E2 -9968.562} C_VEL
LIN {X 0,Y 431.47,Z 384.866,A -85,B 0,C 180,E1 -9969.5,E2 -9969.5} C_VEL
LIN {X 0,Y 430.348,Z 397.651,A -85,B 0,C 180,E1 -9970.59,E2 -9970.59} C_VEL
LIN {X 0,Y 429.286,Z 402.468,A -85,B 0,C 180,E1 -9971.025,E2 -9971.025} C_VEL
LIN {X 0,Y 425.734,Z 410.143,A -85,B 0,C 180,E1 -9971.724,E2 -9971.724} C_VEL
LIN {X 0,Y 422.194,Z 417.499,A -85,B 0,C 180,E1 -9972.488,E2 -9972.488} C_VEL
LIN {X 0,Y 421.139,Z 421.713,A -85,B 0,C 180,E1 -9973.03,E2 -9973.03} C_VEL
LIN {X 0,Y 420.158,Z 431.322,A -85,B 0,C 180,E1 -9974.477,E2 -9974.477} C_VEL
LIN {X 0,Y 419.171,Z 440.812,A -85,B 0,C 180,E1 -9976.177,E2 -9976.177} C_VEL
LIN {X 0,Y 418.557,Z 448.712,A -85,B 0,C 180,E1 -9977.884,E2 -9977.884} C_VEL
LIN {X 0,Y 417.817,Z 456.091,A -85,B 0,C 180,E1 -9979.827,E2 -9979.827} C_VEL
LIN {X 0,Y 417.429,Z 461.947,A -85,B 0,C 180,E1 -9981.772,E2 -9981.772} C_VEL
LIN {X 0,Y 417.194,Z 466.363,A -85,B 0,C 180,E1 -9983.673,E2 -9983.673} C_VEL
LIN {X 0,Y 417.103,Z 468.93,A -85,B 0,C 180,E1 -9985.167,E2 -9985.167} C_VEL
LIN {X 0,Y 417.022,Z 471.257,A -85,B 0,C 180,E1 -9987.102,E2 -9987.102} C_VEL
LIN {X 0,Y 416.991,Z 472.446,A -85,B 0,C 180,E1 -9989.034,E2 -9989.034} C_VEL
LIN {X 0,Y 416.991,Z 472.463,A -85,B 0,C 180,E1 -9990.966,E2 -9990.966} C_VEL
LIN {X 0,Y 417.022,Z 471.339,A -85,B 0,C 180,E1 -9992.898,E2 -9992.898} C_VEL
LIN {X 0,Y 417.096,Z 469.077,A -85,B 0,C 180,E1 -9994.833,E2 -9994.833} C_VEL
LIN {X 0,Y 417.173,Z 465.622,A -85,B 0,C 180,E1 -9996.773,E2 -9996.773} C_VEL
LIN {X 0,Y 417.494,Z 460.891,A -85,B 0,C 180,E1 -9998.714,E2 -9998.714} C_VEL
LIN {X 0,Y 417.911,Z 454.764,A -85,B 0,C 180,E1 -10000.66,E2 -10000.66} C_VEL
LIN {X 0,Y 418.546,Z 448.105,A -85,B 0,C 180,E1 -10002.362,E2 -10002.362} C_VEL
LIN {X 0,Y 419.222,Z 440.062,A -85,B 0,C 180,E1 -10004.069,E2 -10004.069} C_VEL
LIN {X 0,Y 420.242,Z 430.413,A -85,B 0,C 180,E1 -10005.769,E2 -10005.769} C_VEL
LIN {X 0,Y 421.298,Z 420.549,A -85,B 0,C 180,E1 -10007.224,E2 -10007.224} C_VEL
LIN {X 0,Y 422.512,Z 408.821,A -85,B 0,C 180,E1 -10008.675,E2 -10008.675} C_VEL
LIN {X 0,Y 423.841,Z 395.86,A -85,B 0,C 180,E1 -10009.999,E2 -10009.999} C_VEL
LIN {X 0,Y 425.023,Z 382.99,A -85,B 0,C 180,E1 -10011.079,E2 -10011.079} C_VEL
LIN {X 0,Y 426.219,Z 368.875,A -85,B 0,C 180,E1 -10012.032,E2 -10012.032} C_VEL
LIN {X 0,Y 427.189,Z 354.35,A -85,B 0,C 180,E1 -10012.801,E2 -10012.801} C_VEL
LIN {X 0,Y 427.944,Z 339.893,A -85,B 0,C 180,E1 -10013.373,E2 -10013.373} C_VEL
LIN {X 0,Y 428.491,Z 325.862,A -85,B 0,C 180,E1 -10013.758,E2 -10013.758} C_VEL
LIN {X 0,Y 430.894,Z 191.647,A -85,B 0,C 180,E1 -10016.053,E2 -10016.053} C_VEL
LIN {X 0,Y 426.729,Z 172.12,A -85,B 0,C 180,E1 -10016.687,E2 -10016.687} C_VEL
LIN {X 0,Y 422.533,Z 162.055,A -85,B 0,C 180,E1 -10017.191,E2 -10017.191} C_VEL
LIN {X 0,Y 419.893,Z 150.779,A -85,B 0,C 180,E1 -10019.5,E2 -10019.5} C_VEL
LIN {X 0,Y 418.274,Z 144.3,A -85,B 0,C 180,E1 -10020.925,E2 -10020.925} C_VEL
LIN {X 0,Y 418.202,Z 143.999,A -85,B 0,C 180,E1 -10021.397,E2 -10021.397} C_VEL
LIN {X 0,Y 418.253,Z 144.01,A -85,B 0,C 180,E1 -10024.577,E2 -10024.577} C_VEL
LIN {X 0,Y 418.217,Z 144.016,A -85,B 0,C 180,E1 -10027.831,E2 -10027.831} C_VEL
LIN {X 0,Y 418.207,Z 144.01,A -85,B 0,C 180,E1 -10030.95,E2 -10030.95} C_VEL
LIN {X 0,Y 418.202,Z 144.002,A -85,B 0,C 180,E1 -10033.728,E2 -10033.728} C_VEL
LIN {X 0,Y 418.2,Z 144.017,A -85,B 0,C 180,E1 -10036.447,E2 -10036.447} C_VEL
LIN {X 0,Y 418.207,Z 143.991,A -85,B 0,C 180,E1 -10039.133,E2 -10039.133} C_VEL
LIN {X 0,Y 418.238,Z 144.011,A -85,B 0,C 180,E1 -10042.776,E2 -10042.776} C_VEL
LIN {X 0,Y 418.234,Z 143.989,A -85,B 0,C 180,E1 -10046.321,E2 -10046.321} C_VEL
LIN {X 0,Y 418.241,Z 143.993,A -85,B 0,C 180,E1 -10049.727,E2 -10049.727} C_VEL
LIN {X 0,Y 418.213,Z 144.013,A -85,B 0,C 180,E1 -10053.017,E2 -10053.017} C_VEL
LIN {X 0,Y 418.261,Z 144.005,A -85,B 0,C 180,E1 -10056.217,E2 -10056.217} C_VEL
LIN {X 0,Y 418.251,Z 144.003,A -85,B 0,C 180,E1 -10059.337,E2 -10059.337} C_VEL
LIN {X 0,Y 418.258,Z 144.01,A -85,B 0,C 180,E1 -10062.395,E2 -10062.395} C_VEL
LIN {X 0,Y 418.281,Z 143.995,A -85,B 0,C 180,E1 -10065.402,E2 -10065.402} C_VEL
LIN {X 0,Y 418.316,Z 144.002,A -85,B 0,C 180,E1 -10068.369,E2 -10068.369} C_VEL
LIN {X 0,Y 418.379,Z 143.983,A -85,B 0,C 180,E1 -10071.304,E2 -10071.304} C_VEL
LIN {X 0,Y 418.5,Z 143.979,A -85,B 0,C 180,E1 -10074.217,E2 -10074.217} C_VEL
LIN {X 0,Y 418.538,Z 143.963,A -85,B 0,C 180,E1 -10078.075,E2 -10078.075} C_VEL
LIN {X 0,Y 418.666,Z 143.957,A -85,B 0,C 180,E1 -10080,E2 -10080} C_VEL
LIN {X 0,Y 418.494,Z 143.971,A -85,B 0,C 180,E1 -10082.888,E2 -10082.888} C_VEL
LIN {X 0,Y 418.501,Z 143.978,A -85,B 0,C 180,E1 -10085.783,E2 -10085.783} C_VEL
LIN {X 0,Y 418.38,Z 143.988,A -85,B 0,C 180,E1 -10088.695,E2 -10088.695} C_VEL
LIN {X 0,Y 418.317,Z 144.002,A -85,B 0,C 180,E1 -10091.631,E2 -10091.631} C_VEL
LIN {X 0,Y 418.303,Z 143.999,A -85,B 0,C 180,E1 -10094.597,E2 -10094.597} C_VEL
LIN {X 0,Y 418.281,Z 144.006,A -85,B 0,C 180,E1 -10097.604,E2 -10097.604} C_VEL
LIN {X 0,Y 418.251,Z 144.002,A -85,B 0,C 180,E1 -10100.663,E2 -10100.663} C_VEL
LIN {X 0,Y 418.275,Z 144.005,A -85,B 0,C 180,E1 -10103.782,E2 -10103.782} C_VEL
LIN {X 0,Y 418.312,Z 144,A -85,B 0,C 180,E1 -10107.07,E2 -10107.07} C_VEL
LIN {X 0,Y 418.246,Z 144.004,A -85,B 0,C 180,E1 -10110.272,E2 -10110.272} C_VEL
LIN {X 0,Y 418.233,Z 143.98,A -85,B 0,C 180,E1 -10113.678,E2 -10113.678} C_VEL
LIN {X 0,Y 418.241,Z 144.01,A -85,B 0,C 180,E1 -10117.224,E2 -10117.224} C_VEL
LIN {X 0,Y 418.249,Z 143.991,A -85,B 0,C 180,E1 -10119.682,E2 -10119.682} C_VEL
LIN {X 0,Y 418.23,Z 144.007,A -85,B 0,C 180,E1 -10122.321,E2 -10122.321} C_VEL
LIN {X 0,Y 418.236,Z 144.002,A -85,B 0,C 180,E1 -10125.109,E2 -10125.109} C_VEL
LIN {X 0,Y 418.241,Z 144.009,A -85,B 0,C 180,E1 -10127.767,E2 -10127.767} C_VEL
